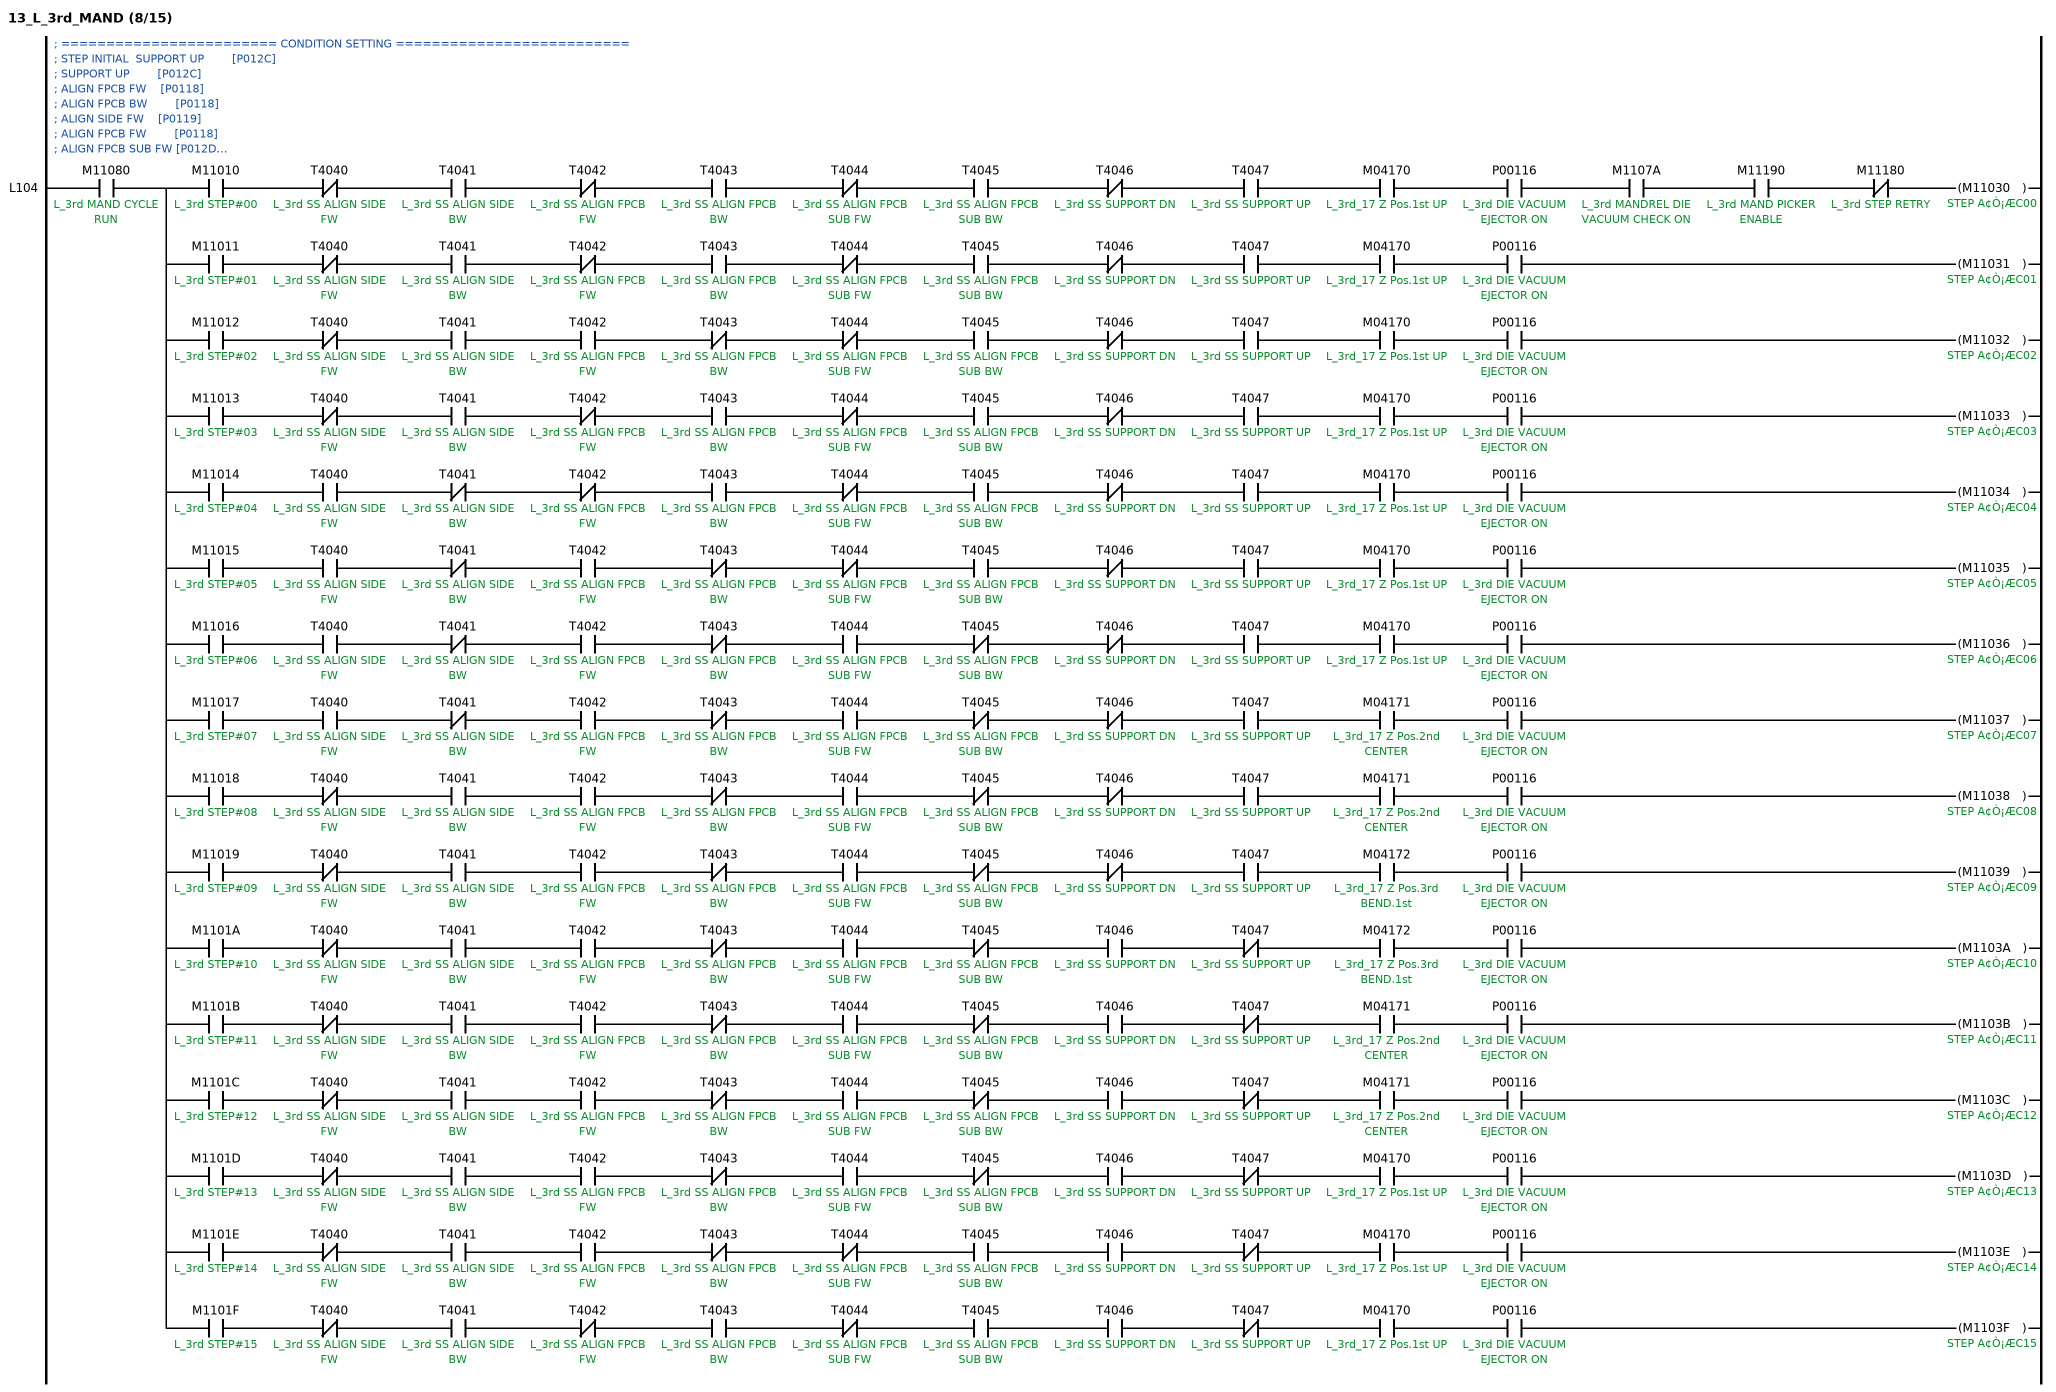
[picture p96: 13_L_3rd_MAND rungs L104-L104]
// ======================== CONDITION SETTING ==========================
; L104
LOAD      M11080	// L_3rd MAND CYCLE RUN
MPUSH
AND       M11010	// L_3rd STEP#00
AND NOT   T4040	// L_3rd SS ALIGN SIDE FW
AND       T4041	// L_3rd SS ALIGN SIDE BW
AND NOT   T4042	// L_3rd SS ALIGN FPCB FW
AND       T4043	// L_3rd SS ALIGN FPCB BW
AND NOT   T4044	// L_3rd SS ALIGN FPCB SUB FW
AND       T4045	// L_3rd SS ALIGN FPCB SUB BW
AND NOT   T4046	// L_3rd SS SUPPORT DN
AND       T4047	// L_3rd SS SUPPORT UP
AND       M04170	// L_3rd_17 Z Pos.1st UP
AND       P00116	// L_3rd DIE VACUUM EJECTOR ON
AND       M1107A	// L_3rd MANDREL DIE VACUUM CHECK ON
AND       M11190	// L_3rd MAND PICKER ENABLE
AND NOT   M11180	// L_3rd STEP RETRY
OUT       M11030	// STEP A¢Ò¡ÆC00
MLOAD
AND       M11011	// L_3rd STEP#01
AND NOT   T4040	// L_3rd SS ALIGN SIDE FW
AND       T4041	// L_3rd SS ALIGN SIDE BW
AND NOT   T4042	// L_3rd SS ALIGN FPCB FW
AND       T4043	// L_3rd SS ALIGN FPCB BW
AND NOT   T4044	// L_3rd SS ALIGN FPCB SUB FW
AND       T4045	// L_3rd SS ALIGN FPCB SUB BW
AND NOT   T4046	// L_3rd SS SUPPORT DN
AND       T4047	// L_3rd SS SUPPORT UP
AND       M04170	// L_3rd_17 Z Pos.1st UP
AND       P00116	// L_3rd DIE VACUUM EJECTOR ON
OUT       M11031	// STEP A¢Ò¡ÆC01
MLOAD
AND       M11012	// L_3rd STEP#02
AND NOT   T4040	// L_3rd SS ALIGN SIDE FW
AND       T4041	// L_3rd SS ALIGN SIDE BW
AND       T4042	// L_3rd SS ALIGN FPCB FW
AND NOT   T4043	// L_3rd SS ALIGN FPCB BW
AND NOT   T4044	// L_3rd SS ALIGN FPCB SUB FW
AND       T4045	// L_3rd SS ALIGN FPCB SUB BW
AND NOT   T4046	// L_3rd SS SUPPORT DN
AND       T4047	// L_3rd SS SUPPORT UP
AND       M04170	// L_3rd_17 Z Pos.1st UP
AND       P00116	// L_3rd DIE VACUUM EJECTOR ON
OUT       M11032	// STEP A¢Ò¡ÆC02
MLOAD
AND       M11013	// L_3rd STEP#03
AND NOT   T4040	// L_3rd SS ALIGN SIDE FW
AND       T4041	// L_3rd SS ALIGN SIDE BW
AND NOT   T4042	// L_3rd SS ALIGN FPCB FW
AND       T4043	// L_3rd SS ALIGN FPCB BW
AND NOT   T4044	// L_3rd SS ALIGN FPCB SUB FW
AND       T4045	// L_3rd SS ALIGN FPCB SUB BW
AND NOT   T4046	// L_3rd SS SUPPORT DN
AND       T4047	// L_3rd SS SUPPORT UP
AND       M04170	// L_3rd_17 Z Pos.1st UP
AND       P00116	// L_3rd DIE VACUUM EJECTOR ON
OUT       M11033	// STEP A¢Ò¡ÆC03
MLOAD
AND       M11014	// L_3rd STEP#04
AND       T4040	// L_3rd SS ALIGN SIDE FW
AND NOT   T4041	// L_3rd SS ALIGN SIDE BW
AND NOT   T4042	// L_3rd SS ALIGN FPCB FW
AND       T4043	// L_3rd SS ALIGN FPCB BW
AND NOT   T4044	// L_3rd SS ALIGN FPCB SUB FW
AND       T4045	// L_3rd SS ALIGN FPCB SUB BW
AND NOT   T4046	// L_3rd SS SUPPORT DN
AND       T4047	// L_3rd SS SUPPORT UP
AND       M04170	// L_3rd_17 Z Pos.1st UP
AND       P00116	// L_3rd DIE VACUUM EJECTOR ON
OUT       M11034	// STEP A¢Ò¡ÆC04
MLOAD
AND       M11015	// L_3rd STEP#05
AND       T4040	// L_3rd SS ALIGN SIDE FW
AND NOT   T4041	// L_3rd SS ALIGN SIDE BW
AND       T4042	// L_3rd SS ALIGN FPCB FW
AND NOT   T4043	// L_3rd SS ALIGN FPCB BW
AND NOT   T4044	// L_3rd SS ALIGN FPCB SUB FW
AND       T4045	// L_3rd SS ALIGN FPCB SUB BW
AND NOT   T4046	// L_3rd SS SUPPORT DN
AND       T4047	// L_3rd SS SUPPORT UP
AND       M04170	// L_3rd_17 Z Pos.1st UP
AND       P00116	// L_3rd DIE VACUUM EJECTOR ON
OUT       M11035	// STEP A¢Ò¡ÆC05
MLOAD
AND       M11016	// L_3rd STEP#06
AND       T4040	// L_3rd SS ALIGN SIDE FW
AND NOT   T4041	// L_3rd SS ALIGN SIDE BW
AND       T4042	// L_3rd SS ALIGN FPCB FW
AND NOT   T4043	// L_3rd SS ALIGN FPCB BW
AND       T4044	// L_3rd SS ALIGN FPCB SUB FW
AND NOT   T4045	// L_3rd SS ALIGN FPCB SUB BW
AND NOT   T4046	// L_3rd SS SUPPORT DN
AND       T4047	// L_3rd SS SUPPORT UP
AND       M04170	// L_3rd_17 Z Pos.1st UP
AND       P00116	// L_3rd DIE VACUUM EJECTOR ON
OUT       M11036	// STEP A¢Ò¡ÆC06
MLOAD
AND       M11017	// L_3rd STEP#07
AND       T4040	// L_3rd SS ALIGN SIDE FW
AND NOT   T4041	// L_3rd SS ALIGN SIDE BW
AND       T4042	// L_3rd SS ALIGN FPCB FW
AND NOT   T4043	// L_3rd SS ALIGN FPCB BW
AND       T4044	// L_3rd SS ALIGN FPCB SUB FW
AND NOT   T4045	// L_3rd SS ALIGN FPCB SUB BW
AND NOT   T4046	// L_3rd SS SUPPORT DN
AND       T4047	// L_3rd SS SUPPORT UP
AND       M04171	// L_3rd_17 Z Pos.2nd CENTER
AND       P00116	// L_3rd DIE VACUUM EJECTOR ON
OUT       M11037	// STEP A¢Ò¡ÆC07
MLOAD
AND       M11018	// L_3rd STEP#08
AND NOT   T4040	// L_3rd SS ALIGN SIDE FW
AND       T4041	// L_3rd SS ALIGN SIDE BW
AND       T4042	// L_3rd SS ALIGN FPCB FW
AND NOT   T4043	// L_3rd SS ALIGN FPCB BW
AND       T4044	// L_3rd SS ALIGN FPCB SUB FW
AND NOT   T4045	// L_3rd SS ALIGN FPCB SUB BW
AND NOT   T4046	// L_3rd SS SUPPORT DN
AND       T4047	// L_3rd SS SUPPORT UP
AND       M04171	// L_3rd_17 Z Pos.2nd CENTER
AND       P00116	// L_3rd DIE VACUUM EJECTOR ON
OUT       M11038	// STEP A¢Ò¡ÆC08
MLOAD
AND       M11019	// L_3rd STEP#09
AND NOT   T4040	// L_3rd SS ALIGN SIDE FW
AND       T4041	// L_3rd SS ALIGN SIDE BW
AND       T4042	// L_3rd SS ALIGN FPCB FW
AND NOT   T4043	// L_3rd SS ALIGN FPCB BW
AND       T4044	// L_3rd SS ALIGN FPCB SUB FW
AND NOT   T4045	// L_3rd SS ALIGN FPCB SUB BW
AND NOT   T4046	// L_3rd SS SUPPORT DN
AND       T4047	// L_3rd SS SUPPORT UP
AND       M04172	// L_3rd_17 Z Pos.3rd BEND.1st
AND       P00116	// L_3rd DIE VACUUM EJECTOR ON
OUT       M11039	// STEP A¢Ò¡ÆC09
MLOAD
AND       M1101A	// L_3rd STEP#10
AND NOT   T4040	// L_3rd SS ALIGN SIDE FW
AND       T4041	// L_3rd SS ALIGN SIDE BW
AND       T4042	// L_3rd SS ALIGN FPCB FW
AND NOT   T4043	// L_3rd SS ALIGN FPCB BW
AND       T4044	// L_3rd SS ALIGN FPCB SUB FW
AND NOT   T4045	// L_3rd SS ALIGN FPCB SUB BW
AND       T4046	// L_3rd SS SUPPORT DN
AND NOT   T4047	// L_3rd SS SUPPORT UP
AND       M04172	// L_3rd_17 Z Pos.3rd BEND.1st
AND       P00116	// L_3rd DIE VACUUM EJECTOR ON
OUT       M1103A	// STEP A¢Ò¡ÆC10
MLOAD
AND       M1101B	// L_3rd STEP#11
AND NOT   T4040	// L_3rd SS ALIGN SIDE FW
AND       T4041	// L_3rd SS ALIGN SIDE BW
AND       T4042	// L_3rd SS ALIGN FPCB FW
AND NOT   T4043	// L_3rd SS ALIGN FPCB BW
AND       T4044	// L_3rd SS ALIGN FPCB SUB FW
AND NOT   T4045	// L_3rd SS ALIGN FPCB SUB BW
AND       T4046	// L_3rd SS SUPPORT DN
AND NOT   T4047	// L_3rd SS SUPPORT UP
AND       M04171	// L_3rd_17 Z Pos.2nd CENTER
AND       P00116	// L_3rd DIE VACUUM EJECTOR ON
OUT       M1103B	// STEP A¢Ò¡ÆC11
MLOAD
AND       M1101C	// L_3rd STEP#12
AND NOT   T4040	// L_3rd SS ALIGN SIDE FW
AND       T4041	// L_3rd SS ALIGN SIDE BW
AND       T4042	// L_3rd SS ALIGN FPCB FW
AND NOT   T4043	// L_3rd SS ALIGN FPCB BW
AND       T4044	// L_3rd SS ALIGN FPCB SUB FW
AND NOT   T4045	// L_3rd SS ALIGN FPCB SUB BW
AND       T4046	// L_3rd SS SUPPORT DN
AND NOT   T4047	// L_3rd SS SUPPORT UP
AND       M04171	// L_3rd_17 Z Pos.2nd CENTER
AND       P00116	// L_3rd DIE VACUUM EJECTOR ON
OUT       M1103C	// STEP A¢Ò¡ÆC12
MLOAD
AND       M1101D	// L_3rd STEP#13
AND NOT   T4040	// L_3rd SS ALIGN SIDE FW
AND       T4041	// L_3rd SS ALIGN SIDE BW
AND       T4042	// L_3rd SS ALIGN FPCB FW
AND NOT   T4043	// L_3rd SS ALIGN FPCB BW
AND       T4044	// L_3rd SS ALIGN FPCB SUB FW
AND NOT   T4045	// L_3rd SS ALIGN FPCB SUB BW
AND       T4046	// L_3rd SS SUPPORT DN
AND NOT   T4047	// L_3rd SS SUPPORT UP
AND       M04170	// L_3rd_17 Z Pos.1st UP
AND       P00116	// L_3rd DIE VACUUM EJECTOR ON
OUT       M1103D	// STEP A¢Ò¡ÆC13
MLOAD
AND       M1101E	// L_3rd STEP#14
AND NOT   T4040	// L_3rd SS ALIGN SIDE FW
AND       T4041	// L_3rd SS ALIGN SIDE BW
AND       T4042	// L_3rd SS ALIGN FPCB FW
AND NOT   T4043	// L_3rd SS ALIGN FPCB BW
AND NOT   T4044	// L_3rd SS ALIGN FPCB SUB FW
AND       T4045	// L_3rd SS ALIGN FPCB SUB BW
AND       T4046	// L_3rd SS SUPPORT DN
AND NOT   T4047	// L_3rd SS SUPPORT UP
AND       M04170	// L_3rd_17 Z Pos.1st UP
AND       P00116	// L_3rd DIE VACUUM EJECTOR ON
OUT       M1103E	// STEP A¢Ò¡ÆC14
MPOP
AND       M1101F	// L_3rd STEP#15
AND NOT   T4040	// L_3rd SS ALIGN SIDE FW
AND       T4041	// L_3rd SS ALIGN SIDE BW
AND NOT   T4042	// L_3rd SS ALIGN FPCB FW
AND       T4043	// L_3rd SS ALIGN FPCB BW
AND NOT   T4044	// L_3rd SS ALIGN FPCB SUB FW
AND       T4045	// L_3rd SS ALIGN FPCB SUB BW
AND       T4046	// L_3rd SS SUPPORT DN
AND NOT   T4047	// L_3rd SS SUPPORT UP
AND       M04170	// L_3rd_17 Z Pos.1st UP
AND       P00116	// L_3rd DIE VACUUM EJECTOR ON
OUT       M1103F	// STEP A¢Ò¡ÆC15
// output comment: STEP INITIAL  SUPPORT UP        [P012C]
// output comment: SUPPORT UP        [P012C]
// output comment: ALIGN FPCB FW    [P0118]
// output comment: ALIGN FPCB BW        [P0118]
// output comment: ALIGN SIDE FW    [P0119]
// output comment: ALIGN FPCB FW        [P0118]
// output comment: ALIGN FPCB SUB FW [P012D]
// output comment: L_3rd_17 Z Pos.2nd CENTER >
// output comment: ALIGN SIDE BW      [P0119]
// output comment: L_3rd_17 Z Pos.3rd BEND.1st >
// output comment: SUPPORT DN      [P012C]
// output comment: L_3rd_17 Z Pos.2nd CENTER >
// output comment: L_3rd_17 Z Pos.1st      UP >
// output comment: ALIGN FPCB SUB BW [P012D]
// output comment: ALIGN FPCB BW    [P0118]

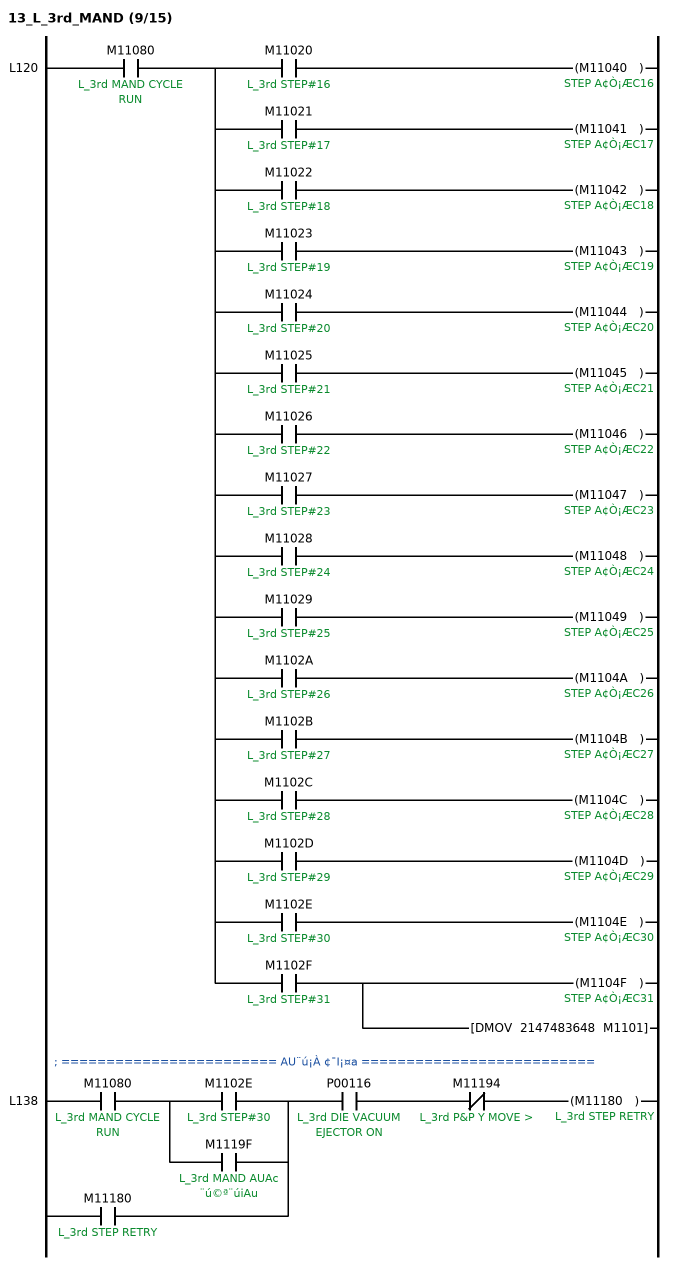
; L120
LOAD      M11080	// L_3rd MAND CYCLE RUN
MPUSH
AND       M11020	// L_3rd STEP#16
OUT       M11040	// STEP A¢Ò¡ÆC16
MLOAD
AND       M11021	// L_3rd STEP#17
OUT       M11041	// STEP A¢Ò¡ÆC17
MLOAD
AND       M11022	// L_3rd STEP#18
OUT       M11042	// STEP A¢Ò¡ÆC18
MLOAD
AND       M11023	// L_3rd STEP#19
OUT       M11043	// STEP A¢Ò¡ÆC19
MLOAD
AND       M11024	// L_3rd STEP#20
OUT       M11044	// STEP A¢Ò¡ÆC20
MLOAD
AND       M11025	// L_3rd STEP#21
OUT       M11045	// STEP A¢Ò¡ÆC21
MLOAD
AND       M11026	// L_3rd STEP#22
OUT       M11046	// STEP A¢Ò¡ÆC22
MLOAD
AND       M11027	// L_3rd STEP#23
OUT       M11047	// STEP A¢Ò¡ÆC23
MLOAD
AND       M11028	// L_3rd STEP#24
OUT       M11048	// STEP A¢Ò¡ÆC24
MLOAD
AND       M11029	// L_3rd STEP#25
OUT       M11049	// STEP A¢Ò¡ÆC25
MLOAD
AND       M1102A	// L_3rd STEP#26
OUT       M1104A	// STEP A¢Ò¡ÆC26
MLOAD
AND       M1102B	// L_3rd STEP#27
OUT       M1104B	// STEP A¢Ò¡ÆC27
MLOAD
AND       M1102C	// L_3rd STEP#28
OUT       M1104C	// STEP A¢Ò¡ÆC28
MLOAD
AND       M1102D	// L_3rd STEP#29
OUT       M1104D	// STEP A¢Ò¡ÆC29
MLOAD
AND       M1102E	// L_3rd STEP#30
OUT       M1104E	// STEP A¢Ò¡ÆC30
MPOP
AND       M1102F	// L_3rd STEP#31
OUT       M1104F	// STEP A¢Ò¡ÆC31
DMOV      2147483648 M1101
// ======================== AU¨ú¡À ¢¯I¡¤a ==========================
; L138
LOAD      M11080	// L_3rd MAND CYCLE RUN
LOAD      M1102E	// L_3rd STEP#30
OR        M1119F	// L_3rd MAND AUAc ¨ú©ª¨úiAu
AND LOAD
OR        M11180	// L_3rd STEP RETRY
AND       P00116	// L_3rd DIE VACUUM EJECTOR ON
AND NOT   M11194	// L_3rd P&P Y MOVE >
OUT       M11180	// L_3rd STEP RETRY

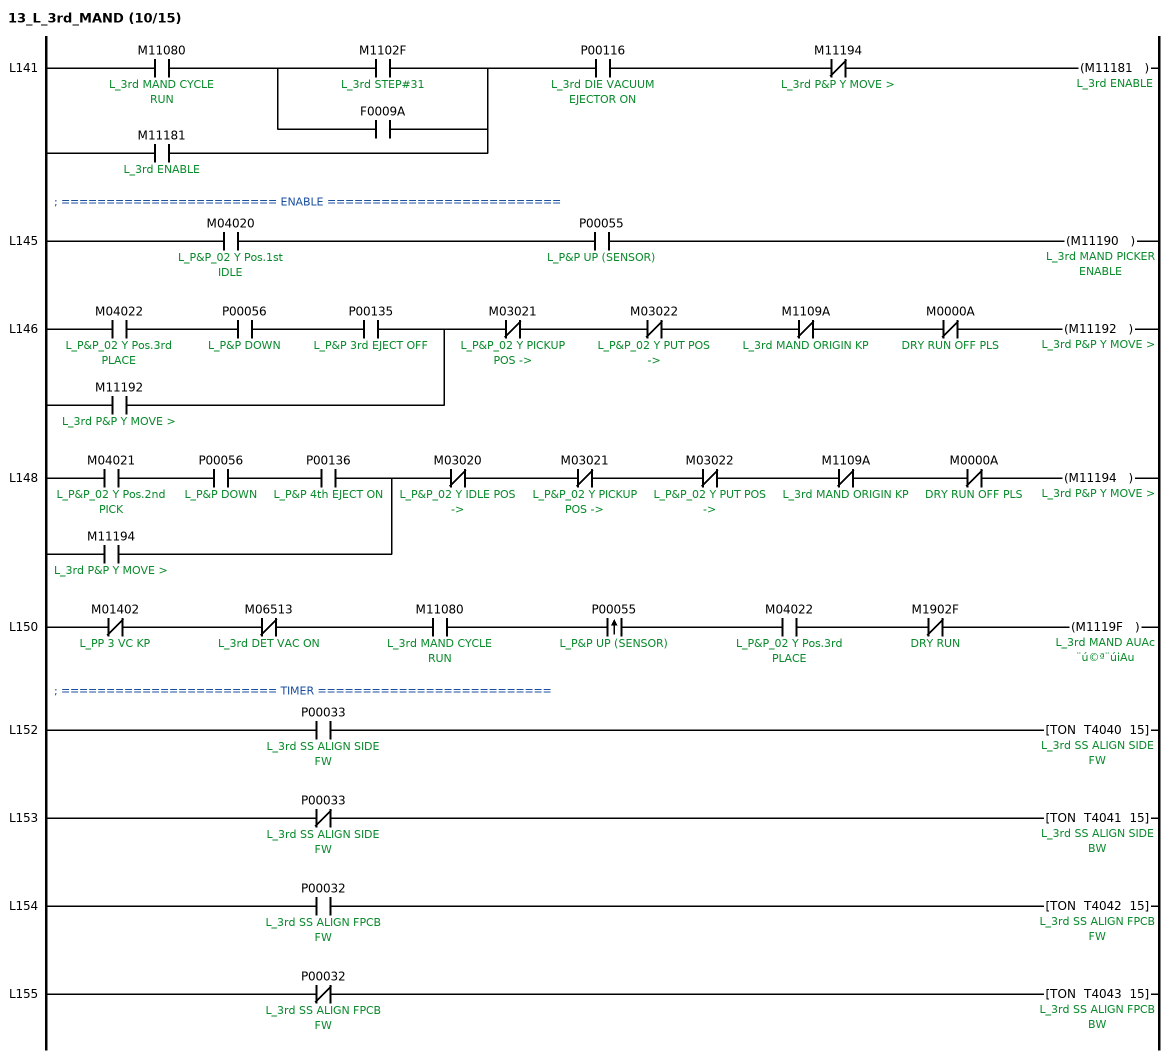
; L141
LOAD      M11080	// L_3rd MAND CYCLE RUN
LOAD      M1102F	// L_3rd STEP#31
OR        F0009A
AND LOAD
OR        M11181	// L_3rd ENABLE
AND       P00116	// L_3rd DIE VACUUM EJECTOR ON
AND NOT   M11194	// L_3rd P&P Y MOVE >
OUT       M11181	// L_3rd ENABLE
// ======================== ENABLE ==========================
; L145
LOAD      M04020	// L_P&P_02 Y Pos.1st IDLE
AND       P00055	// L_P&P UP (SENSOR)
OUT       M11190	// L_3rd MAND PICKER ENABLE
; L146
LOAD      M04022	// L_P&P_02 Y Pos.3rd PLACE
AND       P00056	// L_P&P DOWN
AND       P00135	// L_P&P 3rd EJECT OFF
OR        M11192	// L_3rd P&P Y MOVE >
AND NOT   M03021	// L_P&P_02 Y PICKUP POS ->
AND NOT   M03022	// L_P&P_02 Y PUT POS ->
AND NOT   M1109A	// L_3rd MAND ORIGIN KP
AND NOT   M0000A	// DRY RUN OFF PLS
OUT       M11192	// L_3rd P&P Y MOVE >
; L148
LOAD      M04021	// L_P&P_02 Y Pos.2nd PICK
AND       P00056	// L_P&P DOWN
AND       P00136	// L_P&P 4th EJECT ON
OR        M11194	// L_3rd P&P Y MOVE >
AND NOT   M03020	// L_P&P_02 Y IDLE POS ->
AND NOT   M03021	// L_P&P_02 Y PICKUP POS ->
AND NOT   M03022	// L_P&P_02 Y PUT POS ->
AND NOT   M1109A	// L_3rd MAND ORIGIN KP
AND NOT   M0000A	// DRY RUN OFF PLS
OUT       M11194	// L_3rd P&P Y MOVE >
; L150
LOAD NOT  M01402	// L_PP 3 VC KP
AND NOT   M06513	// L_3rd DET VAC ON
AND       M11080	// L_3rd MAND CYCLE RUN
ANDP      P00055	// L_P&P UP (SENSOR)
AND       M04022	// L_P&P_02 Y Pos.3rd PLACE
AND NOT   M1902F	// DRY RUN
OUT       M1119F	// L_3rd MAND AUAc ¨ú©ª¨úiAu
// ======================== TIMER ==========================
; L152
LOAD      P00033	// L_3rd SS ALIGN SIDE FW
TON       T4040 15	// L_3rd SS ALIGN SIDE FW
; L153
LOAD NOT  P00033	// L_3rd SS ALIGN SIDE FW
TON       T4041 15	// L_3rd SS ALIGN SIDE BW
; L154
LOAD      P00032	// L_3rd SS ALIGN FPCB FW
TON       T4042 15	// L_3rd SS ALIGN FPCB FW
; L155
LOAD NOT  P00032	// L_3rd SS ALIGN FPCB FW
TON       T4043 15	// L_3rd SS ALIGN FPCB BW

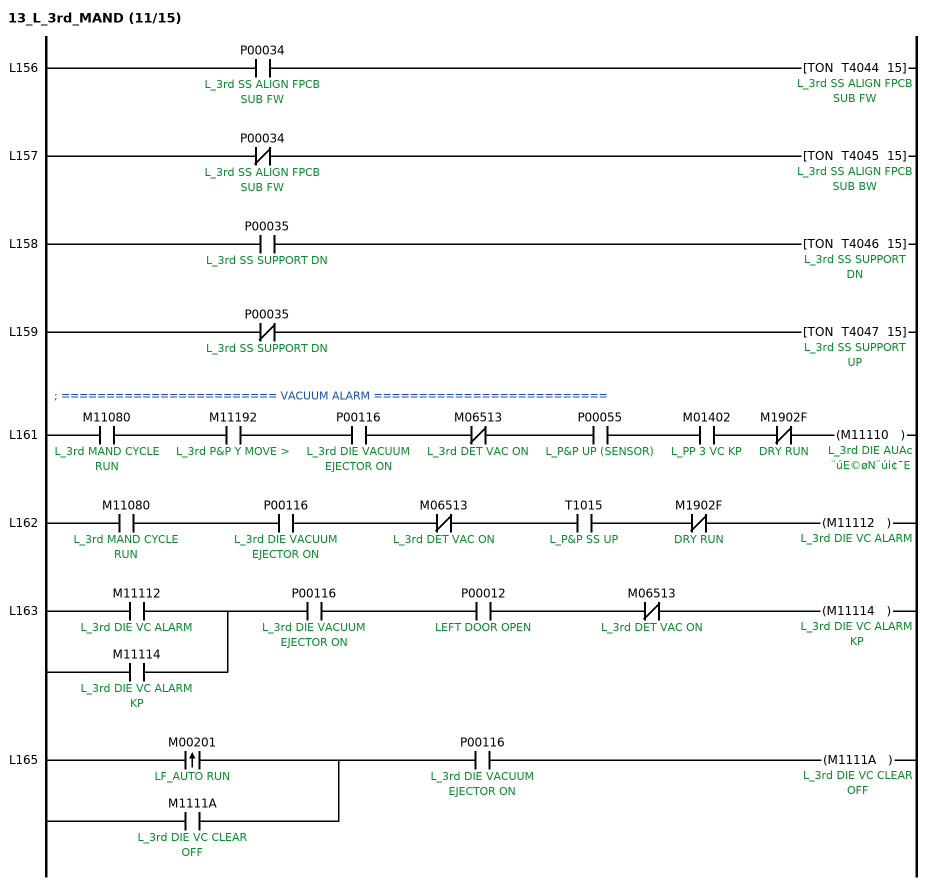
; L156
LOAD      P00034	// L_3rd SS ALIGN FPCB SUB FW
TON       T4044 15	// L_3rd SS ALIGN FPCB SUB FW
; L157
LOAD NOT  P00034	// L_3rd SS ALIGN FPCB SUB FW
TON       T4045 15	// L_3rd SS ALIGN FPCB SUB BW
; L158
LOAD      P00035	// L_3rd SS SUPPORT DN
TON       T4046 15	// L_3rd SS SUPPORT DN
; L159
LOAD NOT  P00035	// L_3rd SS SUPPORT DN
TON       T4047 15	// L_3rd SS SUPPORT UP
// ======================== VACUUM ALARM ==========================
; L161
LOAD      M11080	// L_3rd MAND CYCLE RUN
AND       M11192	// L_3rd P&P Y MOVE >
AND       P00116	// L_3rd DIE VACUUM EJECTOR ON
AND NOT   M06513	// L_3rd DET VAC ON
AND       P00055	// L_P&P UP (SENSOR)
AND       M01402	// L_PP 3 VC KP
AND NOT   M1902F	// DRY RUN
OUT       M11110	// L_3rd DIE AUAc ¨úE©øN¨úi¢¯E
; L162
LOAD      M11080	// L_3rd MAND CYCLE RUN
AND       P00116	// L_3rd DIE VACUUM EJECTOR ON
AND NOT   M06513	// L_3rd DET VAC ON
AND       T1015	// L_P&P SS UP
AND NOT   M1902F	// DRY RUN
OUT       M11112	// L_3rd DIE VC ALARM
; L163
LOAD      M11112	// L_3rd DIE VC ALARM
OR        M11114	// L_3rd DIE VC ALARM KP
AND       P00116	// L_3rd DIE VACUUM EJECTOR ON
AND       P00012	// LEFT DOOR OPEN
AND NOT   M06513	// L_3rd DET VAC ON
OUT       M11114	// L_3rd DIE VC ALARM KP
; L165
LOADP     M00201	// LF_AUTO RUN
OR        M1111A	// L_3rd DIE VC CLEAR OFF
AND       P00116	// L_3rd DIE VACUUM EJECTOR ON
OUT       M1111A	// L_3rd DIE VC CLEAR OFF

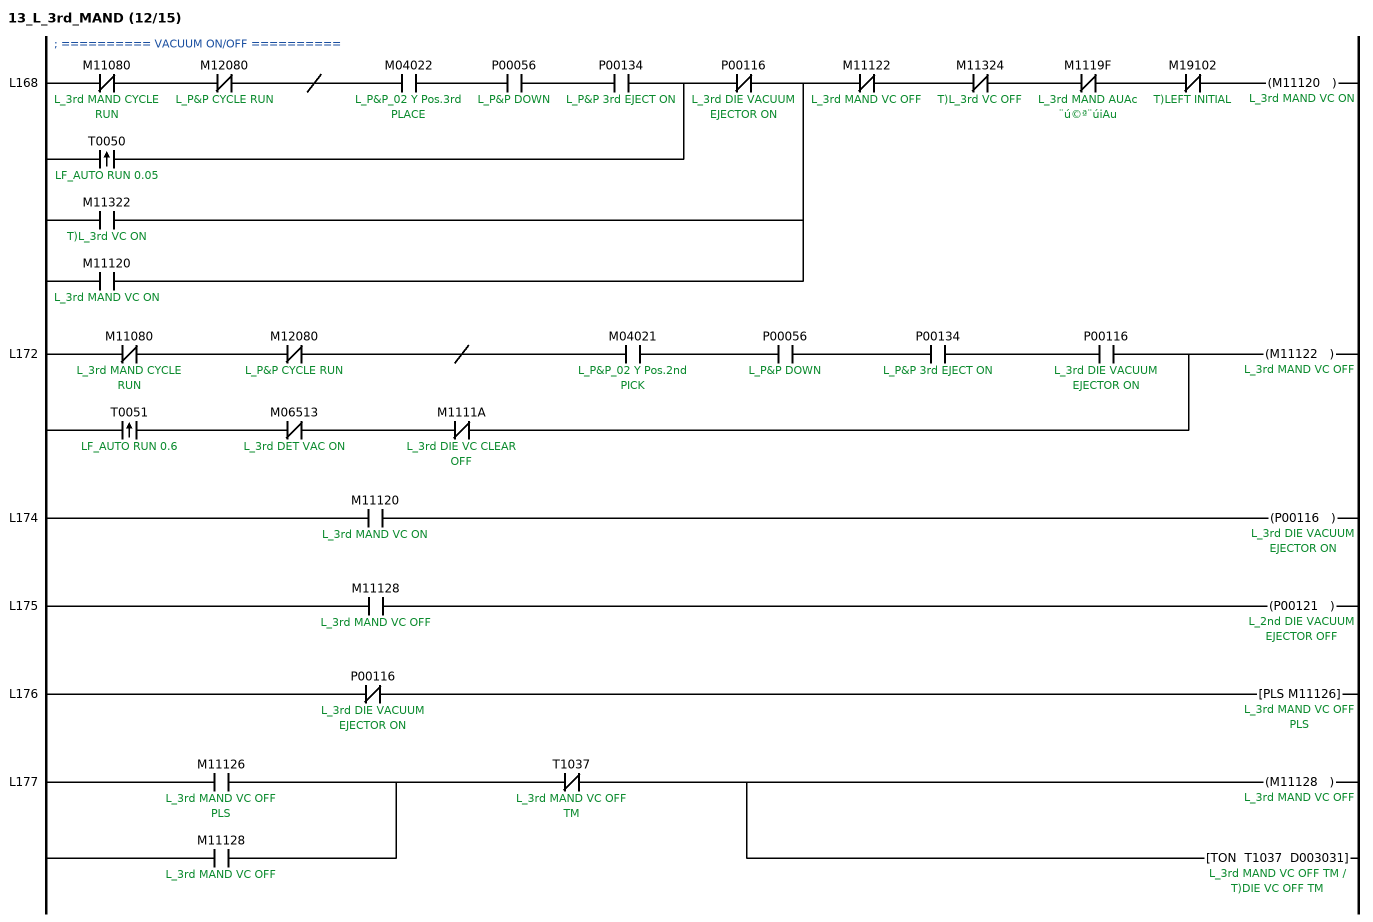
// ========== VACUUM ON/OFF ==========
; L168
LOAD NOT  M11080	// L_3rd MAND CYCLE RUN
AND NOT   M12080	// L_P&P CYCLE RUN
NOT
AND       M04022	// L_P&P_02 Y Pos.3rd PLACE
AND       P00056	// L_P&P DOWN
AND       P00134	// L_P&P 3rd EJECT ON
ORP       T0050	// LF_AUTO RUN 0.05
AND NOT   P00116	// L_3rd DIE VACUUM EJECTOR ON
OR        M11322	// T)L_3rd VC ON
OR        M11120	// L_3rd MAND VC ON
AND NOT   M11122	// L_3rd MAND VC OFF
AND NOT   M11324	// T)L_3rd VC OFF
AND NOT   M1119F	// L_3rd MAND AUAc ¨ú©ª¨úiAu
AND NOT   M19102	// T)LEFT INITIAL
OUT       M11120	// L_3rd MAND VC ON
; L172
LOAD NOT  M11080	// L_3rd MAND CYCLE RUN
AND NOT   M12080	// L_P&P CYCLE RUN
NOT
AND       M04021	// L_P&P_02 Y Pos.2nd PICK
AND       P00056	// L_P&P DOWN
AND       P00134	// L_P&P 3rd EJECT ON
AND       P00116	// L_3rd DIE VACUUM EJECTOR ON
LOADP     T0051	// LF_AUTO RUN 0.6
AND NOT   M06513	// L_3rd DET VAC ON
AND NOT   M1111A	// L_3rd DIE VC CLEAR OFF
OR LOAD
OUT       M11122	// L_3rd MAND VC OFF
; L174
LOAD      M11120	// L_3rd MAND VC ON
OUT       P00116	// L_3rd DIE VACUUM EJECTOR ON
; L175
LOAD      M11128	// L_3rd MAND VC OFF
OUT       P00121	// L_2nd DIE VACUUM EJECTOR OFF
; L176
LOAD NOT  P00116	// L_3rd DIE VACUUM EJECTOR ON
OUTP      M11126	// L_3rd MAND VC OFF PLS
; L177
LOAD      M11126	// L_3rd MAND VC OFF PLS
OR        M11128	// L_3rd MAND VC OFF
AND NOT   T1037	// L_3rd MAND VC OFF TM
OUT       M11128	// L_3rd MAND VC OFF
TON       T1037 D003031	// L_3rd MAND VC OFF TM / T)DIE VC OFF TM

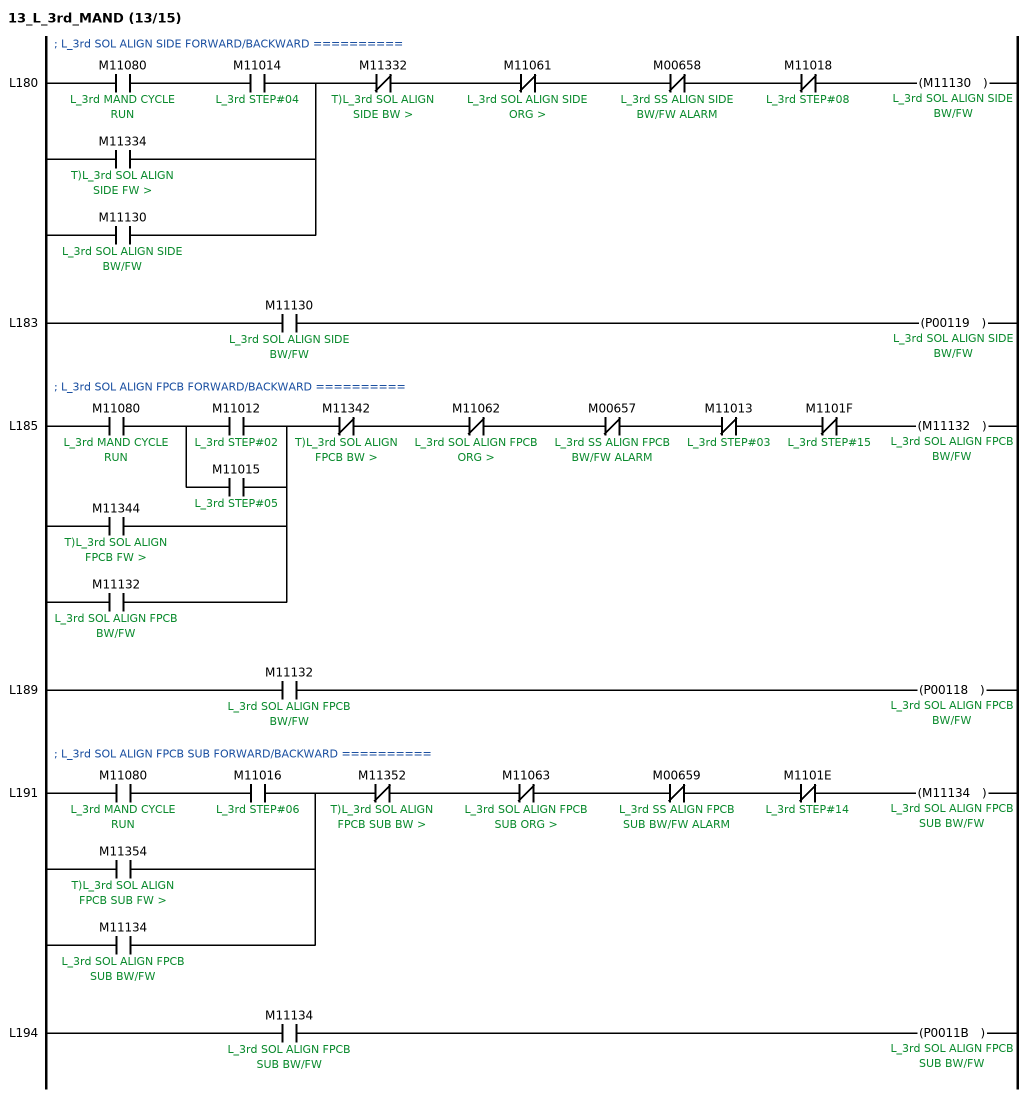
// L_3rd SOL ALIGN SIDE FORWARD/BACKWARD ==========
; L180
LOAD      M11080	// L_3rd MAND CYCLE RUN
AND       M11014	// L_3rd STEP#04
OR        M11334	// T)L_3rd SOL ALIGN SIDE FW >
OR        M11130	// L_3rd SOL ALIGN SIDE BW/FW
AND NOT   M11332	// T)L_3rd SOL ALIGN SIDE BW >
AND NOT   M11061	// L_3rd SOL ALIGN SIDE ORG >
AND NOT   M00658	// L_3rd SS ALIGN SIDE BW/FW ALARM
AND NOT   M11018	// L_3rd STEP#08
OUT       M11130	// L_3rd SOL ALIGN SIDE BW/FW
; L183
LOAD      M11130	// L_3rd SOL ALIGN SIDE BW/FW
OUT       P00119	// L_3rd SOL ALIGN SIDE BW/FW
// L_3rd SOL ALIGN FPCB FORWARD/BACKWARD ==========
; L185
LOAD      M11080	// L_3rd MAND CYCLE RUN
LOAD      M11012	// L_3rd STEP#02
OR        M11015	// L_3rd STEP#05
AND LOAD
OR        M11344	// T)L_3rd SOL ALIGN FPCB FW >
OR        M11132	// L_3rd SOL ALIGN FPCB BW/FW
AND NOT   M11342	// T)L_3rd SOL ALIGN FPCB BW >
AND NOT   M11062	// L_3rd SOL ALIGN FPCB ORG >
AND NOT   M00657	// L_3rd SS ALIGN FPCB BW/FW ALARM
AND NOT   M11013	// L_3rd STEP#03
AND NOT   M1101F	// L_3rd STEP#15
OUT       M11132	// L_3rd SOL ALIGN FPCB BW/FW
; L189
LOAD      M11132	// L_3rd SOL ALIGN FPCB BW/FW
OUT       P00118	// L_3rd SOL ALIGN FPCB BW/FW
// L_3rd SOL ALIGN FPCB SUB FORWARD/BACKWARD ==========
; L191
LOAD      M11080	// L_3rd MAND CYCLE RUN
AND       M11016	// L_3rd STEP#06
OR        M11354	// T)L_3rd SOL ALIGN FPCB SUB FW >
OR        M11134	// L_3rd SOL ALIGN FPCB SUB BW/FW
AND NOT   M11352	// T)L_3rd SOL ALIGN FPCB SUB BW >
AND NOT   M11063	// L_3rd SOL ALIGN FPCB SUB ORG >
AND NOT   M00659	// L_3rd SS ALIGN FPCB SUB BW/FW ALARM
AND NOT   M1101E	// L_3rd STEP#14
OUT       M11134	// L_3rd SOL ALIGN FPCB SUB BW/FW
; L194
LOAD      M11134	// L_3rd SOL ALIGN FPCB SUB BW/FW
OUT       P0011B	// L_3rd SOL ALIGN FPCB SUB BW/FW

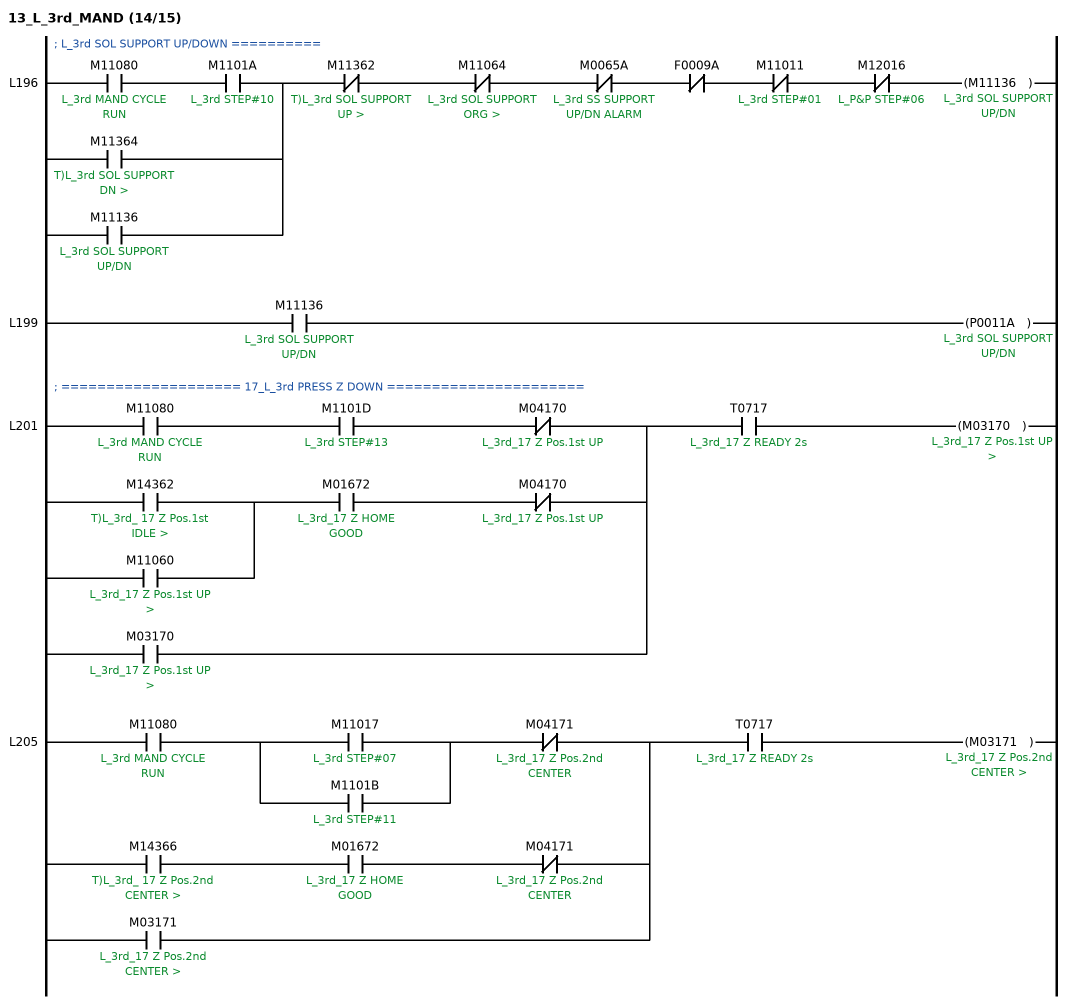
// L_3rd SOL SUPPORT UP/DOWN ==========
; L196
LOAD      M11080	// L_3rd MAND CYCLE RUN
AND       M1101A	// L_3rd STEP#10
OR        M11364	// T)L_3rd SOL SUPPORT DN >
OR        M11136	// L_3rd SOL SUPPORT UP/DN
AND NOT   M11362	// T)L_3rd SOL SUPPORT UP >
AND NOT   M11064	// L_3rd SOL SUPPORT ORG >
AND NOT   M0065A	// L_3rd SS SUPPORT UP/DN ALARM
AND NOT   F0009A
AND NOT   M11011	// L_3rd STEP#01
AND NOT   M12016	// L_P&P STEP#06
OUT       M11136	// L_3rd SOL SUPPORT UP/DN
; L199
LOAD      M11136	// L_3rd SOL SUPPORT UP/DN
OUT       P0011A	// L_3rd SOL SUPPORT UP/DN
// ==================== 17_L_3rd PRESS Z DOWN ======================
; L201
LOAD      M11080	// L_3rd MAND CYCLE RUN
AND       M1101D	// L_3rd STEP#13
AND NOT   M04170	// L_3rd_17 Z Pos.1st UP
LOAD      M14362	// T)L_3rd_ 17 Z Pos.1st IDLE >
OR        M11060	// L_3rd_17 Z Pos.1st UP >
AND       M01672	// L_3rd_17 Z HOME GOOD
AND NOT   M04170	// L_3rd_17 Z Pos.1st UP
OR LOAD
OR        M03170	// L_3rd_17 Z Pos.1st UP >
AND       T0717	// L_3rd_17 Z READY 2s
OUT       M03170	// L_3rd_17 Z Pos.1st UP >
; L205
LOAD      M11080	// L_3rd MAND CYCLE RUN
LOAD      M11017	// L_3rd STEP#07
OR        M1101B	// L_3rd STEP#11
AND LOAD
AND NOT   M04171	// L_3rd_17 Z Pos.2nd CENTER
LOAD      M14366	// T)L_3rd_ 17 Z Pos.2nd CENTER >
AND       M01672	// L_3rd_17 Z HOME GOOD
AND NOT   M04171	// L_3rd_17 Z Pos.2nd CENTER
OR LOAD
OR        M03171	// L_3rd_17 Z Pos.2nd CENTER >
AND       T0717	// L_3rd_17 Z READY 2s
OUT       M03171	// L_3rd_17 Z Pos.2nd CENTER >

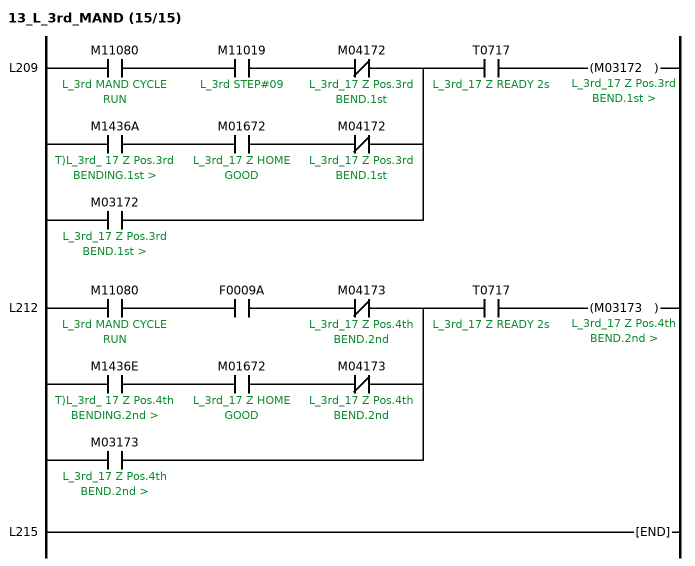
; L209
LOAD      M11080	// L_3rd MAND CYCLE RUN
AND       M11019	// L_3rd STEP#09
AND NOT   M04172	// L_3rd_17 Z Pos.3rd BEND.1st
LOAD      M1436A	// T)L_3rd_ 17 Z Pos.3rd BENDING.1st >
AND       M01672	// L_3rd_17 Z HOME GOOD
AND NOT   M04172	// L_3rd_17 Z Pos.3rd BEND.1st
OR LOAD
OR        M03172	// L_3rd_17 Z Pos.3rd BEND.1st >
AND       T0717	// L_3rd_17 Z READY 2s
OUT       M03172	// L_3rd_17 Z Pos.3rd BEND.1st >
; L212
LOAD      M11080	// L_3rd MAND CYCLE RUN
AND       F0009A
AND NOT   M04173	// L_3rd_17 Z Pos.4th BEND.2nd
LOAD      M1436E	// T)L_3rd_ 17 Z Pos.4th BENDING.2nd >
AND       M01672	// L_3rd_17 Z HOME GOOD
AND NOT   M04173	// L_3rd_17 Z Pos.4th BEND.2nd
OR LOAD
OR        M03173	// L_3rd_17 Z Pos.4th BEND.2nd >
AND       T0717	// L_3rd_17 Z READY 2s
OUT       M03173	// L_3rd_17 Z Pos.4th BEND.2nd >
; L215
END

PROGRAM 14_L_TOOL (task: ½ºÄµ ÇÁ·Î±×·¥)

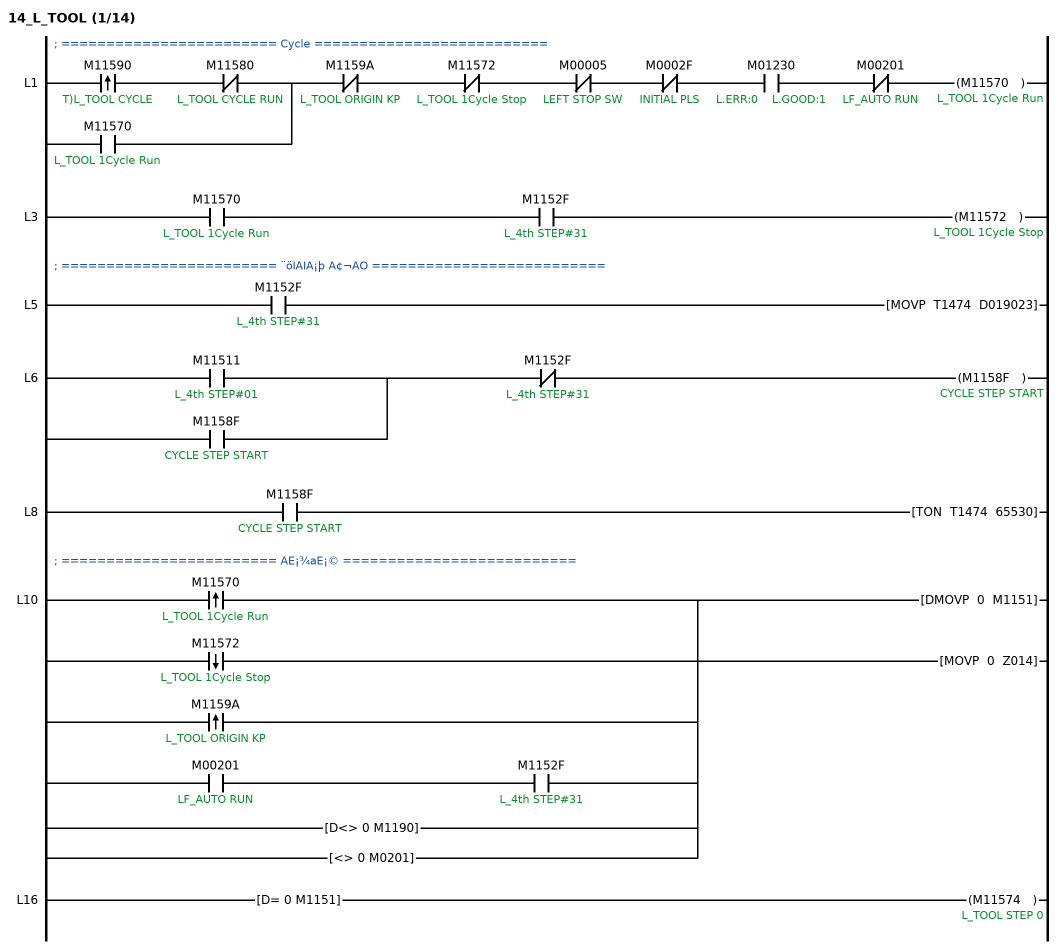
// ======================== Cycle ==========================
; L1
LOADP     M11590	// T)L_TOOL CYCLE
AND NOT   M11580	// L_TOOL CYCLE RUN
OR        M11570	// L_TOOL 1Cycle Run
AND NOT   M1159A	// L_TOOL ORIGIN KP
AND NOT   M11572	// L_TOOL 1Cycle Stop
AND NOT   M00005	// LEFT STOP SW
AND NOT   M0002F	// INITIAL PLS
AND       M01230	// L.ERR:0    L.GOOD:1
AND NOT   M00201	// LF_AUTO RUN
OUT       M11570	// L_TOOL 1Cycle Run
; L3
LOAD      M11570	// L_TOOL 1Cycle Run
AND       M1152F	// L_4th STEP#31
OUT       M11572	// L_TOOL 1Cycle Stop
// ======================== ¨öIAIA¡þ A¢¬AO ==========================
; L5
LOAD      M1152F	// L_4th STEP#31
MOVP      T1474 D019023
; L6
LOAD      M11511	// L_4th STEP#01
OR        M1158F	// CYCLE STEP START
AND NOT   M1152F	// L_4th STEP#31
OUT       M1158F	// CYCLE STEP START
; L8
LOAD      M1158F	// CYCLE STEP START
TON       T1474 65530
// ======================== AE¡¾aE¡© ==========================
; L10
LOADP     M11570	// L_TOOL 1Cycle Run
ORN       M11572	// L_TOOL 1Cycle Stop
ORP       M1159A	// L_TOOL ORIGIN KP
LOAD      M00201	// LF_AUTO RUN
AND       M1152F	// L_4th STEP#31
OR LOAD
ORD<>     0 M1190
OR<>      0 M0201
DMOVP     0 M1151
MOVP      0 Z014
; L16
LOADD=    0 M1151
OUT       M11574	// L_TOOL STEP 0

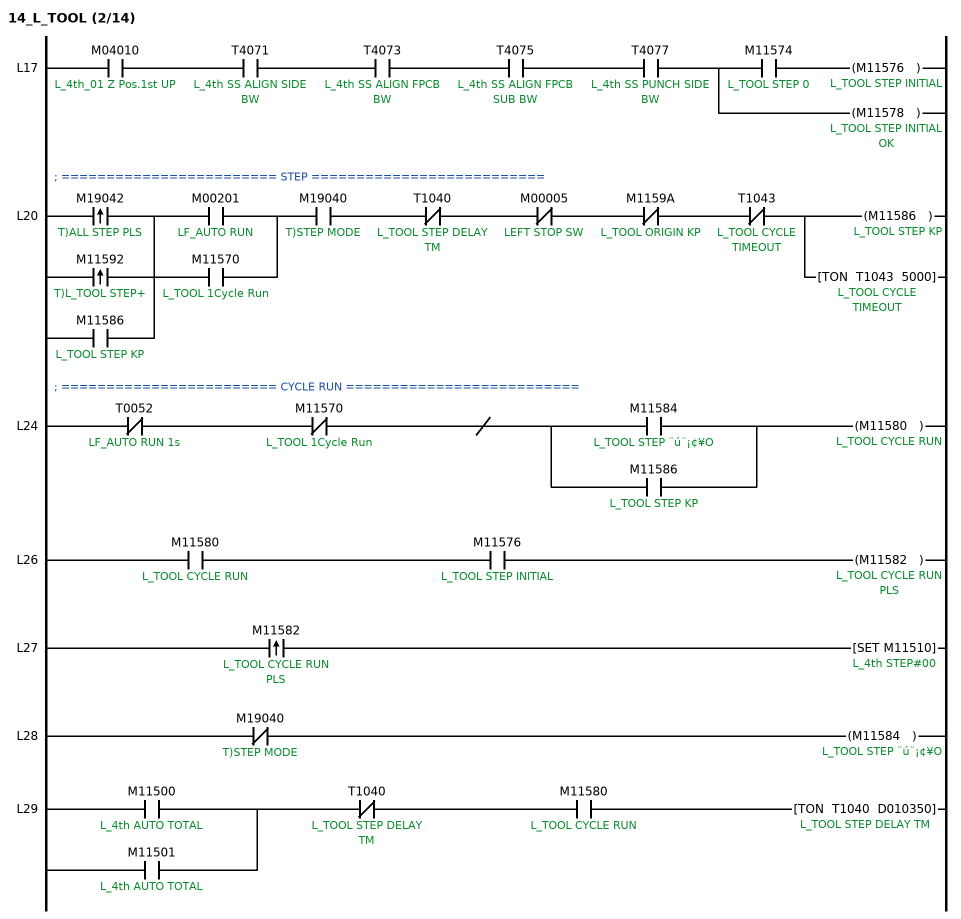
; L17
LOAD      M04010	// L_4th_01 Z Pos.1st UP
AND       T4071	// L_4th SS ALIGN SIDE BW
AND       T4073	// L_4th SS ALIGN FPCB BW
AND       T4075	// L_4th SS ALIGN FPCB SUB BW
AND       T4077	// L_4th SS PUNCH SIDE BW
MPUSH
AND       M11574	// L_TOOL STEP 0
OUT       M11576	// L_TOOL STEP INITIAL
MPOP
OUT       M11578	// L_TOOL STEP INITIAL OK
// ======================== STEP ==========================
; L20
LOADP     M19042	// T)ALL STEP PLS
ORP       M11592	// T)L_TOOL STEP+
OR        M11586	// L_TOOL STEP KP
LOAD      M00201	// LF_AUTO RUN
OR        M11570	// L_TOOL 1Cycle Run
AND LOAD
AND       M19040	// T)STEP MODE
AND NOT   T1040	// L_TOOL STEP DELAY TM
AND NOT   M00005	// LEFT STOP SW
AND NOT   M1159A	// L_TOOL ORIGIN KP
AND NOT   T1043	// L_TOOL CYCLE TIMEOUT
OUT       M11586	// L_TOOL STEP KP
TON       T1043 5000	// L_TOOL CYCLE TIMEOUT
// ======================== CYCLE RUN ==========================
; L24
LOAD NOT  T0052	// LF_AUTO RUN 1s
AND NOT   M11570	// L_TOOL 1Cycle Run
NOT
LOAD      M11584	// L_TOOL STEP ¨ú¨¡¢¥O
OR        M11586	// L_TOOL STEP KP
AND LOAD
OUT       M11580	// L_TOOL CYCLE RUN
; L26
LOAD      M11580	// L_TOOL CYCLE RUN
AND       M11576	// L_TOOL STEP INITIAL
OUT       M11582	// L_TOOL CYCLE RUN PLS
; L27
LOADP     M11582	// L_TOOL CYCLE RUN PLS
SET       M11510	// L_4th STEP#00
; L28
LOAD NOT  M19040	// T)STEP MODE
OUT       M11584	// L_TOOL STEP ¨ú¨¡¢¥O
; L29
LOAD      M11500	// L_4th AUTO TOTAL
OR        M11501	// L_4th AUTO TOTAL
AND NOT   T1040	// L_TOOL STEP DELAY TM
AND       M11580	// L_TOOL CYCLE RUN
TON       T1040 D010350	// L_TOOL STEP DELAY TM

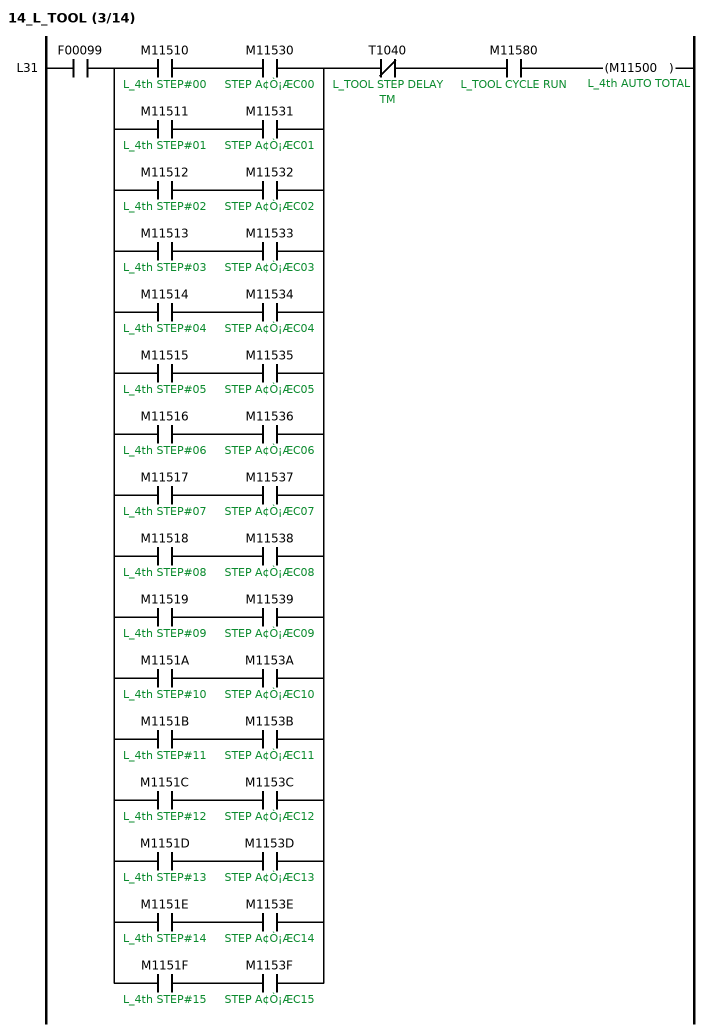
; L31
LOAD      F00099
LOAD      M11510	// L_4th STEP#00
AND       M11530	// STEP A¢Ò¡ÆC00
LOAD      M11511	// L_4th STEP#01
AND       M11531	// STEP A¢Ò¡ÆC01
OR LOAD
LOAD      M11512	// L_4th STEP#02
AND       M11532	// STEP A¢Ò¡ÆC02
OR LOAD
LOAD      M11513	// L_4th STEP#03
AND       M11533	// STEP A¢Ò¡ÆC03
OR LOAD
LOAD      M11514	// L_4th STEP#04
AND       M11534	// STEP A¢Ò¡ÆC04
OR LOAD
LOAD      M11515	// L_4th STEP#05
AND       M11535	// STEP A¢Ò¡ÆC05
OR LOAD
LOAD      M11516	// L_4th STEP#06
AND       M11536	// STEP A¢Ò¡ÆC06
OR LOAD
LOAD      M11517	// L_4th STEP#07
AND       M11537	// STEP A¢Ò¡ÆC07
OR LOAD
LOAD      M11518	// L_4th STEP#08
AND       M11538	// STEP A¢Ò¡ÆC08
OR LOAD
LOAD      M11519	// L_4th STEP#09
AND       M11539	// STEP A¢Ò¡ÆC09
OR LOAD
LOAD      M1151A	// L_4th STEP#10
AND       M1153A	// STEP A¢Ò¡ÆC10
OR LOAD
LOAD      M1151B	// L_4th STEP#11
AND       M1153B	// STEP A¢Ò¡ÆC11
OR LOAD
LOAD      M1151C	// L_4th STEP#12
AND       M1153C	// STEP A¢Ò¡ÆC12
OR LOAD
LOAD      M1151D	// L_4th STEP#13
AND       M1153D	// STEP A¢Ò¡ÆC13
OR LOAD
LOAD      M1151E	// L_4th STEP#14
AND       M1153E	// STEP A¢Ò¡ÆC14
OR LOAD
LOAD      M1151F	// L_4th STEP#15
AND       M1153F	// STEP A¢Ò¡ÆC15
OR LOAD
AND LOAD
AND NOT   T1040	// L_TOOL STEP DELAY TM
AND       M11580	// L_TOOL CYCLE RUN
OUT       M11500	// L_4th AUTO TOTAL

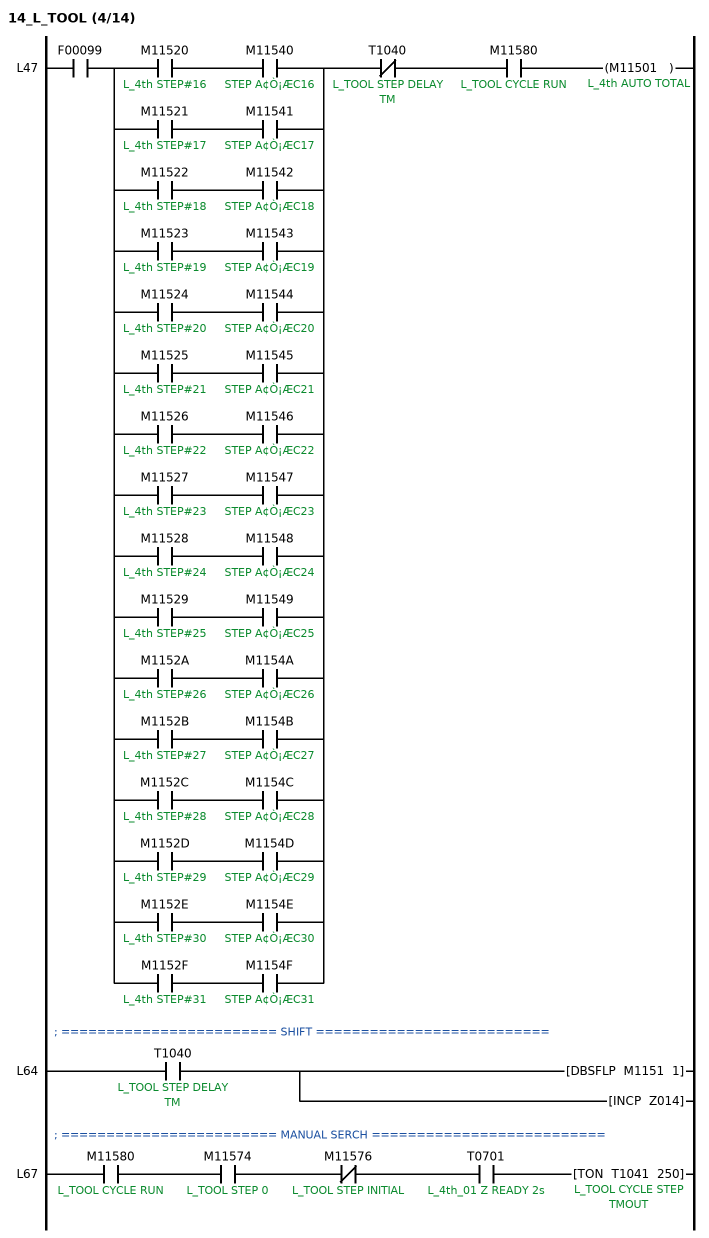
; L47
LOAD      F00099
LOAD      M11520	// L_4th STEP#16
AND       M11540	// STEP A¢Ò¡ÆC16
LOAD      M11521	// L_4th STEP#17
AND       M11541	// STEP A¢Ò¡ÆC17
OR LOAD
LOAD      M11522	// L_4th STEP#18
AND       M11542	// STEP A¢Ò¡ÆC18
OR LOAD
LOAD      M11523	// L_4th STEP#19
AND       M11543	// STEP A¢Ò¡ÆC19
OR LOAD
LOAD      M11524	// L_4th STEP#20
AND       M11544	// STEP A¢Ò¡ÆC20
OR LOAD
LOAD      M11525	// L_4th STEP#21
AND       M11545	// STEP A¢Ò¡ÆC21
OR LOAD
LOAD      M11526	// L_4th STEP#22
AND       M11546	// STEP A¢Ò¡ÆC22
OR LOAD
LOAD      M11527	// L_4th STEP#23
AND       M11547	// STEP A¢Ò¡ÆC23
OR LOAD
LOAD      M11528	// L_4th STEP#24
AND       M11548	// STEP A¢Ò¡ÆC24
OR LOAD
LOAD      M11529	// L_4th STEP#25
AND       M11549	// STEP A¢Ò¡ÆC25
OR LOAD
LOAD      M1152A	// L_4th STEP#26
AND       M1154A	// STEP A¢Ò¡ÆC26
OR LOAD
LOAD      M1152B	// L_4th STEP#27
AND       M1154B	// STEP A¢Ò¡ÆC27
OR LOAD
LOAD      M1152C	// L_4th STEP#28
AND       M1154C	// STEP A¢Ò¡ÆC28
OR LOAD
LOAD      M1152D	// L_4th STEP#29
AND       M1154D	// STEP A¢Ò¡ÆC29
OR LOAD
LOAD      M1152E	// L_4th STEP#30
AND       M1154E	// STEP A¢Ò¡ÆC30
OR LOAD
LOAD      M1152F	// L_4th STEP#31
AND       M1154F	// STEP A¢Ò¡ÆC31
OR LOAD
AND LOAD
AND NOT   T1040	// L_TOOL STEP DELAY TM
AND       M11580	// L_TOOL CYCLE RUN
OUT       M11501	// L_4th AUTO TOTAL
// ======================== SHIFT ==========================
; L64
LOAD      T1040	// L_TOOL STEP DELAY TM
DBSFLP    M1151 1
INCP      Z014
// ======================== MANUAL SERCH ==========================
; L67
LOAD      M11580	// L_TOOL CYCLE RUN
AND       M11574	// L_TOOL STEP 0
AND NOT   M11576	// L_TOOL STEP INITIAL
AND       T0701	// L_4th_01 Z READY 2s
TON       T1041 250	// L_TOOL CYCLE STEP TMOUT

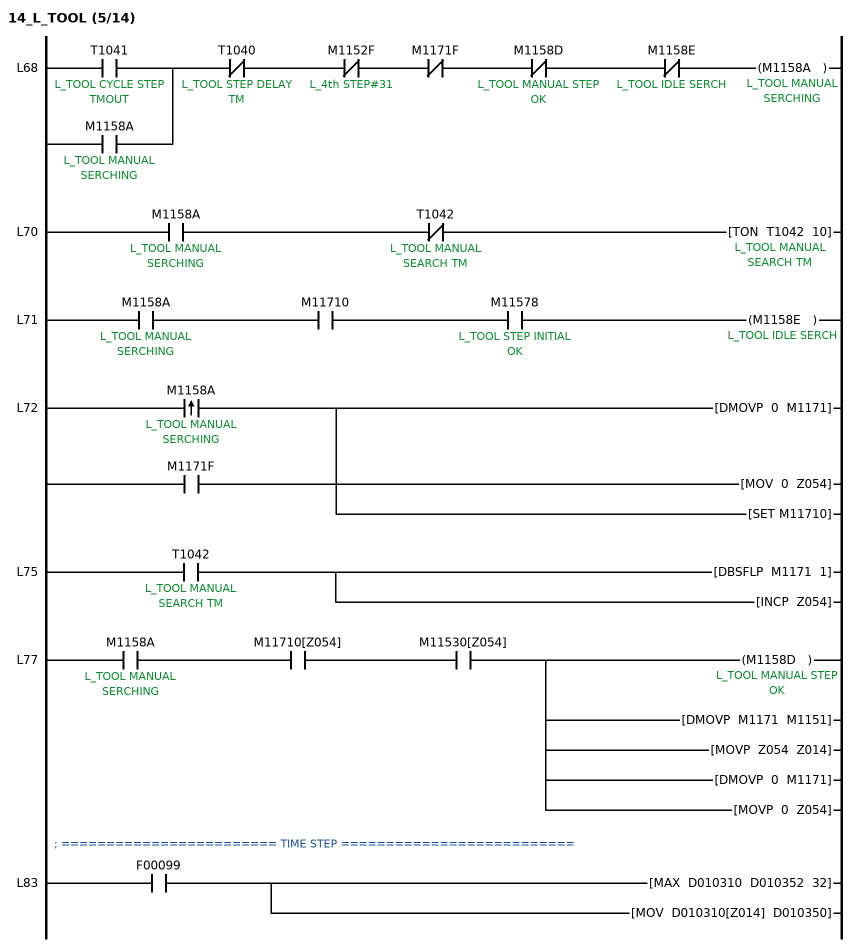
; L68
LOAD      T1041	// L_TOOL CYCLE STEP TMOUT
OR        M1158A	// L_TOOL MANUAL SERCHING
AND NOT   T1040	// L_TOOL STEP DELAY TM
AND NOT   M1152F	// L_4th STEP#31
AND NOT   M1171F
AND NOT   M1158D	// L_TOOL MANUAL STEP OK
AND NOT   M1158E	// L_TOOL IDLE SERCH
OUT       M1158A	// L_TOOL MANUAL SERCHING
; L70
LOAD      M1158A	// L_TOOL MANUAL SERCHING
AND NOT   T1042	// L_TOOL MANUAL SEARCH TM
TON       T1042 10	// L_TOOL MANUAL SEARCH TM
; L71
LOAD      M1158A	// L_TOOL MANUAL SERCHING
AND       M11710
AND       M11578	// L_TOOL STEP INITIAL OK
OUT       M1158E	// L_TOOL IDLE SERCH
; L72
LOADP     M1158A	// L_TOOL MANUAL SERCHING
OR        M1171F
DMOVP     0 M1171
MOV       0 Z054
SET       M11710
; L75
LOAD      T1042	// L_TOOL MANUAL SEARCH TM
DBSFLP    M1171 1
INCP      Z054
; L77
LOAD      M1158A	// L_TOOL MANUAL SERCHING
AND       M11710[Z054]
AND       M11530[Z054]
OUT       M1158D	// L_TOOL MANUAL STEP OK
DMOVP     M1171 M1151
MOVP      Z054 Z014
DMOVP     0 M1171
MOVP      0 Z054
// ======================== TIME STEP ==========================
; L83
LOAD      F00099
MAX       D010310 D010352 32
MOV       D010310[Z014] D010350

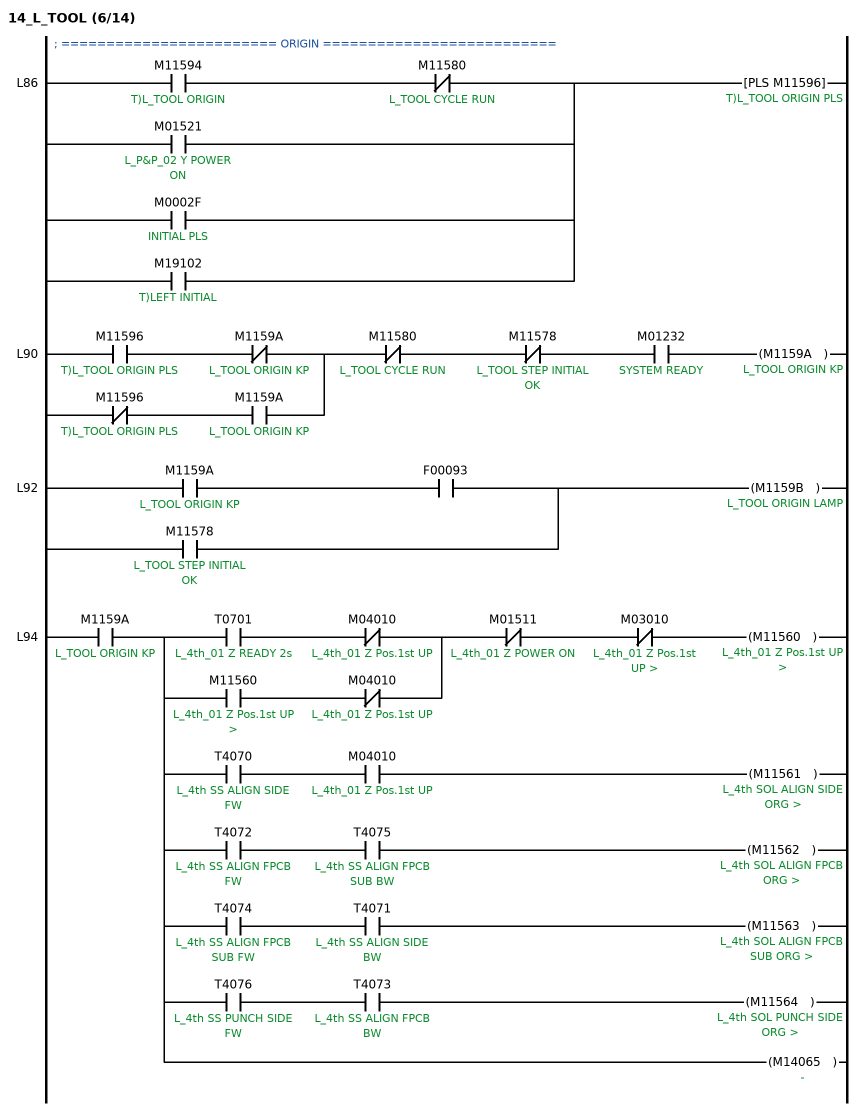
// ======================== ORIGIN ==========================
; L86
LOAD      M11594	// T)L_TOOL ORIGIN
AND NOT   M11580	// L_TOOL CYCLE RUN
OR        M01521	// L_P&P_02 Y POWER ON
OR        M0002F	// INITIAL PLS
OR        M19102	// T)LEFT INITIAL
OUTP      M11596	// T)L_TOOL ORIGIN PLS
; L90
LOAD      M11596	// T)L_TOOL ORIGIN PLS
AND NOT   M1159A	// L_TOOL ORIGIN KP
LOAD NOT  M11596	// T)L_TOOL ORIGIN PLS
AND       M1159A	// L_TOOL ORIGIN KP
OR LOAD
AND NOT   M11580	// L_TOOL CYCLE RUN
AND NOT   M11578	// L_TOOL STEP INITIAL OK
AND       M01232	// SYSTEM READY
OUT       M1159A	// L_TOOL ORIGIN KP
; L92
LOAD      M1159A	// L_TOOL ORIGIN KP
AND       F00093
OR        M11578	// L_TOOL STEP INITIAL OK
OUT       M1159B	// L_TOOL ORIGIN LAMP
; L94
LOAD      M1159A	// L_TOOL ORIGIN KP
MPUSH
LOAD      T0701	// L_4th_01 Z READY 2s
AND NOT   M04010	// L_4th_01 Z Pos.1st UP
LOAD      M11560	// L_4th_01 Z Pos.1st UP >
AND NOT   M04010	// L_4th_01 Z Pos.1st UP
OR LOAD
AND LOAD
AND NOT   M01511	// L_4th_01 Z POWER ON
AND NOT   M03010	// L_4th_01 Z Pos.1st     UP >
OUT       M11560	// L_4th_01 Z Pos.1st UP >
MLOAD
AND       T4070	// L_4th SS ALIGN SIDE FW
AND       M04010	// L_4th_01 Z Pos.1st UP
OUT       M11561	// L_4th SOL ALIGN SIDE ORG >
MLOAD
AND       T4072	// L_4th SS ALIGN FPCB FW
AND       T4075	// L_4th SS ALIGN FPCB SUB BW
OUT       M11562	// L_4th SOL ALIGN FPCB ORG >
MLOAD
AND       T4074	// L_4th SS ALIGN FPCB SUB FW
AND       T4071	// L_4th SS ALIGN SIDE BW
OUT       M11563	// L_4th SOL ALIGN FPCB SUB ORG >
MLOAD
AND       T4076	// L_4th SS PUNCH SIDE FW
AND       T4073	// L_4th SS ALIGN FPCB BW
OUT       M11564	// L_4th SOL PUNCH SIDE ORG >
MPOP
OUT       M14065	// -

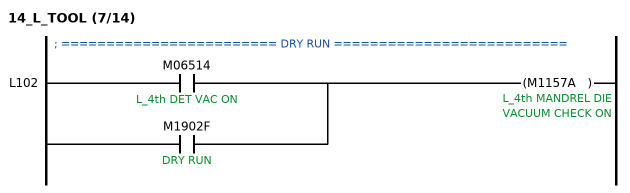
// ======================== DRY RUN ==========================
; L102
LOAD      M06514	// L_4th DET VAC ON
OR        M1902F	// DRY RUN
OUT       M1157A	// L_4th MANDREL DIE VACUUM CHECK ON

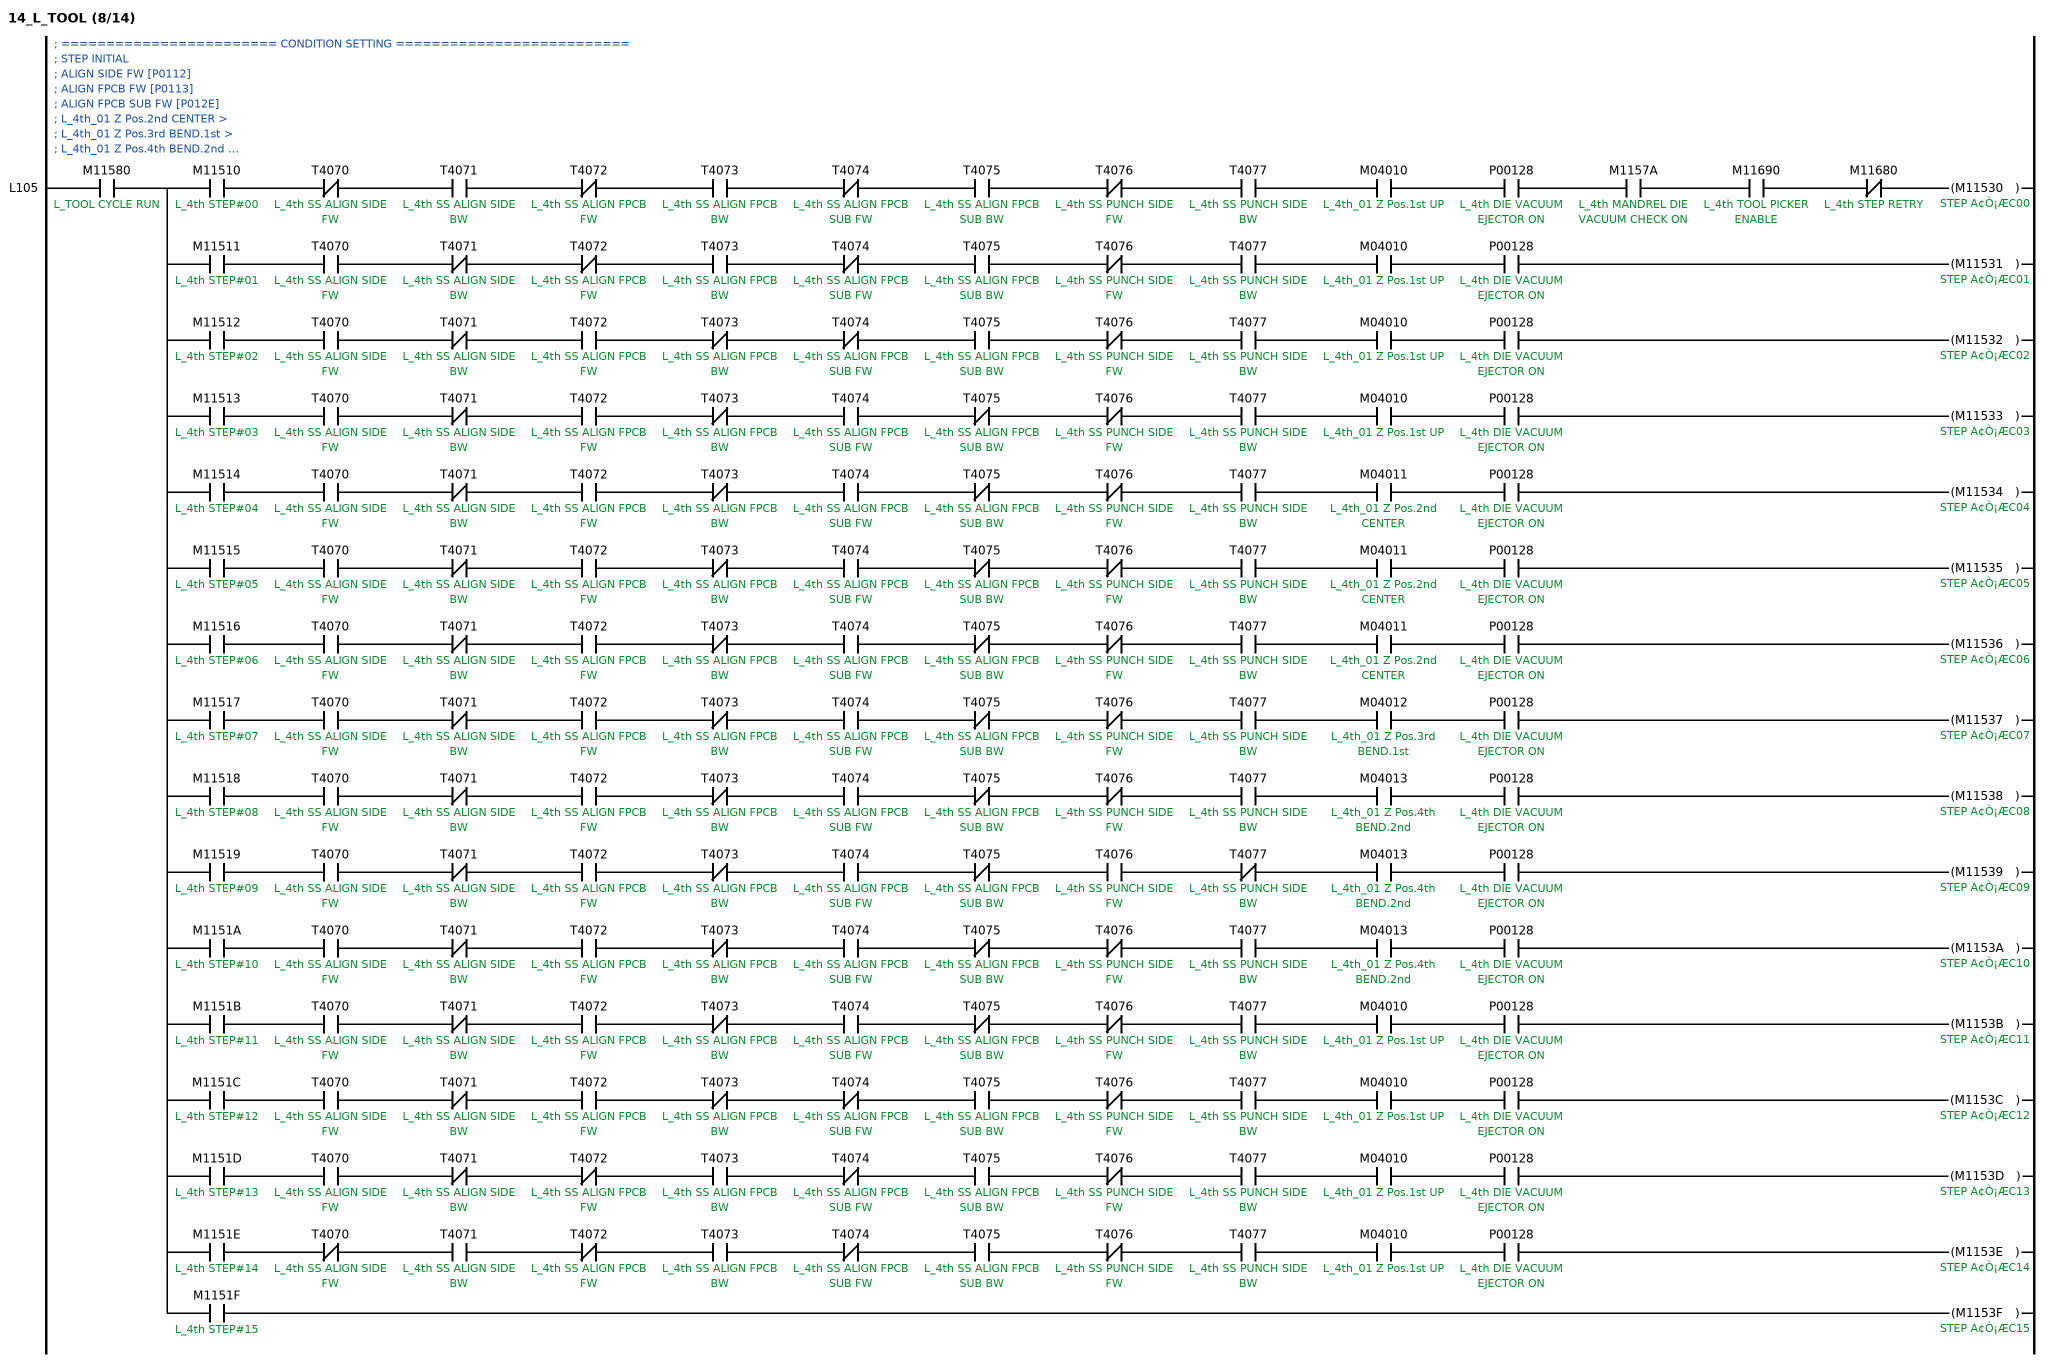
// ======================== CONDITION SETTING ==========================
; L105
LOAD      M11580	// L_TOOL CYCLE RUN
MPUSH
AND       M11510	// L_4th STEP#00
AND NOT   T4070	// L_4th SS ALIGN SIDE FW
AND       T4071	// L_4th SS ALIGN SIDE BW
AND NOT   T4072	// L_4th SS ALIGN FPCB FW
AND       T4073	// L_4th SS ALIGN FPCB BW
AND NOT   T4074	// L_4th SS ALIGN FPCB SUB FW
AND       T4075	// L_4th SS ALIGN FPCB SUB BW
AND NOT   T4076	// L_4th SS PUNCH SIDE FW
AND       T4077	// L_4th SS PUNCH SIDE BW
AND       M04010	// L_4th_01 Z Pos.1st UP
AND       P00128	// L_4th DIE VACUUM EJECTOR ON
AND       M1157A	// L_4th MANDREL DIE VACUUM CHECK ON
AND       M11690	// L_4th TOOL PICKER ENABLE
AND NOT   M11680	// L_4th STEP RETRY
OUT       M11530	// STEP A¢Ò¡ÆC00
MLOAD
AND       M11511	// L_4th STEP#01
AND       T4070	// L_4th SS ALIGN SIDE FW
AND NOT   T4071	// L_4th SS ALIGN SIDE BW
AND NOT   T4072	// L_4th SS ALIGN FPCB FW
AND       T4073	// L_4th SS ALIGN FPCB BW
AND NOT   T4074	// L_4th SS ALIGN FPCB SUB FW
AND       T4075	// L_4th SS ALIGN FPCB SUB BW
AND NOT   T4076	// L_4th SS PUNCH SIDE FW
AND       T4077	// L_4th SS PUNCH SIDE BW
AND       M04010	// L_4th_01 Z Pos.1st UP
AND       P00128	// L_4th DIE VACUUM EJECTOR ON
OUT       M11531	// STEP A¢Ò¡ÆC01
MLOAD
AND       M11512	// L_4th STEP#02
AND       T4070	// L_4th SS ALIGN SIDE FW
AND NOT   T4071	// L_4th SS ALIGN SIDE BW
AND       T4072	// L_4th SS ALIGN FPCB FW
AND NOT   T4073	// L_4th SS ALIGN FPCB BW
AND NOT   T4074	// L_4th SS ALIGN FPCB SUB FW
AND       T4075	// L_4th SS ALIGN FPCB SUB BW
AND NOT   T4076	// L_4th SS PUNCH SIDE FW
AND       T4077	// L_4th SS PUNCH SIDE BW
AND       M04010	// L_4th_01 Z Pos.1st UP
AND       P00128	// L_4th DIE VACUUM EJECTOR ON
OUT       M11532	// STEP A¢Ò¡ÆC02
MLOAD
AND       M11513	// L_4th STEP#03
AND       T4070	// L_4th SS ALIGN SIDE FW
AND NOT   T4071	// L_4th SS ALIGN SIDE BW
AND       T4072	// L_4th SS ALIGN FPCB FW
AND NOT   T4073	// L_4th SS ALIGN FPCB BW
AND       T4074	// L_4th SS ALIGN FPCB SUB FW
AND NOT   T4075	// L_4th SS ALIGN FPCB SUB BW
AND NOT   T4076	// L_4th SS PUNCH SIDE FW
AND       T4077	// L_4th SS PUNCH SIDE BW
AND       M04010	// L_4th_01 Z Pos.1st UP
AND       P00128	// L_4th DIE VACUUM EJECTOR ON
OUT       M11533	// STEP A¢Ò¡ÆC03
MLOAD
AND       M11514	// L_4th STEP#04
AND       T4070	// L_4th SS ALIGN SIDE FW
AND NOT   T4071	// L_4th SS ALIGN SIDE BW
AND       T4072	// L_4th SS ALIGN FPCB FW
AND NOT   T4073	// L_4th SS ALIGN FPCB BW
AND       T4074	// L_4th SS ALIGN FPCB SUB FW
AND NOT   T4075	// L_4th SS ALIGN FPCB SUB BW
AND NOT   T4076	// L_4th SS PUNCH SIDE FW
AND       T4077	// L_4th SS PUNCH SIDE BW
AND       M04011	// L_4th_01 Z Pos.2nd CENTER
AND       P00128	// L_4th DIE VACUUM EJECTOR ON
OUT       M11534	// STEP A¢Ò¡ÆC04
MLOAD
AND       M11515	// L_4th STEP#05
AND       T4070	// L_4th SS ALIGN SIDE FW
AND NOT   T4071	// L_4th SS ALIGN SIDE BW
AND       T4072	// L_4th SS ALIGN FPCB FW
AND NOT   T4073	// L_4th SS ALIGN FPCB BW
AND       T4074	// L_4th SS ALIGN FPCB SUB FW
AND NOT   T4075	// L_4th SS ALIGN FPCB SUB BW
AND NOT   T4076	// L_4th SS PUNCH SIDE FW
AND       T4077	// L_4th SS PUNCH SIDE BW
AND       M04011	// L_4th_01 Z Pos.2nd CENTER
AND       P00128	// L_4th DIE VACUUM EJECTOR ON
OUT       M11535	// STEP A¢Ò¡ÆC05
MLOAD
AND       M11516	// L_4th STEP#06
AND       T4070	// L_4th SS ALIGN SIDE FW
AND NOT   T4071	// L_4th SS ALIGN SIDE BW
AND       T4072	// L_4th SS ALIGN FPCB FW
AND NOT   T4073	// L_4th SS ALIGN FPCB BW
AND       T4074	// L_4th SS ALIGN FPCB SUB FW
AND NOT   T4075	// L_4th SS ALIGN FPCB SUB BW
AND NOT   T4076	// L_4th SS PUNCH SIDE FW
AND       T4077	// L_4th SS PUNCH SIDE BW
AND       M04011	// L_4th_01 Z Pos.2nd CENTER
AND       P00128	// L_4th DIE VACUUM EJECTOR ON
OUT       M11536	// STEP A¢Ò¡ÆC06
MLOAD
AND       M11517	// L_4th STEP#07
AND       T4070	// L_4th SS ALIGN SIDE FW
AND NOT   T4071	// L_4th SS ALIGN SIDE BW
AND       T4072	// L_4th SS ALIGN FPCB FW
AND NOT   T4073	// L_4th SS ALIGN FPCB BW
AND       T4074	// L_4th SS ALIGN FPCB SUB FW
AND NOT   T4075	// L_4th SS ALIGN FPCB SUB BW
AND NOT   T4076	// L_4th SS PUNCH SIDE FW
AND       T4077	// L_4th SS PUNCH SIDE BW
AND       M04012	// L_4th_01 Z Pos.3rd BEND.1st
AND       P00128	// L_4th DIE VACUUM EJECTOR ON
OUT       M11537	// STEP A¢Ò¡ÆC07
MLOAD
AND       M11518	// L_4th STEP#08
AND       T4070	// L_4th SS ALIGN SIDE FW
AND NOT   T4071	// L_4th SS ALIGN SIDE BW
AND       T4072	// L_4th SS ALIGN FPCB FW
AND NOT   T4073	// L_4th SS ALIGN FPCB BW
AND       T4074	// L_4th SS ALIGN FPCB SUB FW
AND NOT   T4075	// L_4th SS ALIGN FPCB SUB BW
AND NOT   T4076	// L_4th SS PUNCH SIDE FW
AND       T4077	// L_4th SS PUNCH SIDE BW
AND       M04013	// L_4th_01 Z Pos.4th BEND.2nd
AND       P00128	// L_4th DIE VACUUM EJECTOR ON
OUT       M11538	// STEP A¢Ò¡ÆC08
MLOAD
AND       M11519	// L_4th STEP#09
AND       T4070	// L_4th SS ALIGN SIDE FW
AND NOT   T4071	// L_4th SS ALIGN SIDE BW
AND       T4072	// L_4th SS ALIGN FPCB FW
AND NOT   T4073	// L_4th SS ALIGN FPCB BW
AND       T4074	// L_4th SS ALIGN FPCB SUB FW
AND NOT   T4075	// L_4th SS ALIGN FPCB SUB BW
AND       T4076	// L_4th SS PUNCH SIDE FW
AND NOT   T4077	// L_4th SS PUNCH SIDE BW
AND       M04013	// L_4th_01 Z Pos.4th BEND.2nd
AND       P00128	// L_4th DIE VACUUM EJECTOR ON
OUT       M11539	// STEP A¢Ò¡ÆC09
MLOAD
AND       M1151A	// L_4th STEP#10
AND       T4070	// L_4th SS ALIGN SIDE FW
AND NOT   T4071	// L_4th SS ALIGN SIDE BW
AND       T4072	// L_4th SS ALIGN FPCB FW
AND NOT   T4073	// L_4th SS ALIGN FPCB BW
AND       T4074	// L_4th SS ALIGN FPCB SUB FW
AND NOT   T4075	// L_4th SS ALIGN FPCB SUB BW
AND NOT   T4076	// L_4th SS PUNCH SIDE FW
AND       T4077	// L_4th SS PUNCH SIDE BW
AND       M04013	// L_4th_01 Z Pos.4th BEND.2nd
AND       P00128	// L_4th DIE VACUUM EJECTOR ON
OUT       M1153A	// STEP A¢Ò¡ÆC10
MLOAD
AND       M1151B	// L_4th STEP#11
AND       T4070	// L_4th SS ALIGN SIDE FW
AND NOT   T4071	// L_4th SS ALIGN SIDE BW
AND       T4072	// L_4th SS ALIGN FPCB FW
AND NOT   T4073	// L_4th SS ALIGN FPCB BW
AND       T4074	// L_4th SS ALIGN FPCB SUB FW
AND NOT   T4075	// L_4th SS ALIGN FPCB SUB BW
AND NOT   T4076	// L_4th SS PUNCH SIDE FW
AND       T4077	// L_4th SS PUNCH SIDE BW
AND       M04010	// L_4th_01 Z Pos.1st UP
AND       P00128	// L_4th DIE VACUUM EJECTOR ON
OUT       M1153B	// STEP A¢Ò¡ÆC11
MLOAD
AND       M1151C	// L_4th STEP#12
AND       T4070	// L_4th SS ALIGN SIDE FW
AND NOT   T4071	// L_4th SS ALIGN SIDE BW
AND       T4072	// L_4th SS ALIGN FPCB FW
AND NOT   T4073	// L_4th SS ALIGN FPCB BW
AND NOT   T4074	// L_4th SS ALIGN FPCB SUB FW
AND       T4075	// L_4th SS ALIGN FPCB SUB BW
AND NOT   T4076	// L_4th SS PUNCH SIDE FW
AND       T4077	// L_4th SS PUNCH SIDE BW
AND       M04010	// L_4th_01 Z Pos.1st UP
AND       P00128	// L_4th DIE VACUUM EJECTOR ON
OUT       M1153C	// STEP A¢Ò¡ÆC12
MLOAD
AND       M1151D	// L_4th STEP#13
AND       T4070	// L_4th SS ALIGN SIDE FW
AND NOT   T4071	// L_4th SS ALIGN SIDE BW
AND NOT   T4072	// L_4th SS ALIGN FPCB FW
AND       T4073	// L_4th SS ALIGN FPCB BW
AND NOT   T4074	// L_4th SS ALIGN FPCB SUB FW
AND       T4075	// L_4th SS ALIGN FPCB SUB BW
AND NOT   T4076	// L_4th SS PUNCH SIDE FW
AND       T4077	// L_4th SS PUNCH SIDE BW
AND       M04010	// L_4th_01 Z Pos.1st UP
AND       P00128	// L_4th DIE VACUUM EJECTOR ON
OUT       M1153D	// STEP A¢Ò¡ÆC13
MLOAD
AND       M1151E	// L_4th STEP#14
AND NOT   T4070	// L_4th SS ALIGN SIDE FW
AND       T4071	// L_4th SS ALIGN SIDE BW
AND NOT   T4072	// L_4th SS ALIGN FPCB FW
AND       T4073	// L_4th SS ALIGN FPCB BW
AND NOT   T4074	// L_4th SS ALIGN FPCB SUB FW
AND       T4075	// L_4th SS ALIGN FPCB SUB BW
AND NOT   T4076	// L_4th SS PUNCH SIDE FW
AND       T4077	// L_4th SS PUNCH SIDE BW
AND       M04010	// L_4th_01 Z Pos.1st UP
AND       P00128	// L_4th DIE VACUUM EJECTOR ON
OUT       M1153E	// STEP A¢Ò¡ÆC14
MPOP
AND       M1151F	// L_4th STEP#15
OUT       M1153F	// STEP A¢Ò¡ÆC15
// output comment: STEP INITIAL
// output comment: ALIGN SIDE FW [P0112]
// output comment: ALIGN FPCB FW [P0113]
// output comment: ALIGN FPCB SUB FW [P012E]
// output comment: L_4th_01 Z Pos.2nd CENTER >
// output comment: L_4th_01 Z Pos.3rd BEND.1st >
// output comment: L_4th_01 Z Pos.4th BEND.2nd >
// output comment: PUNCH SIDE FW [P012F]
// output comment: PUNCH SIDE BW [P012F]
// output comment: L_4th_01 Z Pos.1st       UP >
// output comment: ALIGN FPCB SUB BW [P012E]
// output comment: ALIGN FPCB BW [P0113]
// output comment: ALIGN SIDE BW   [P0112]

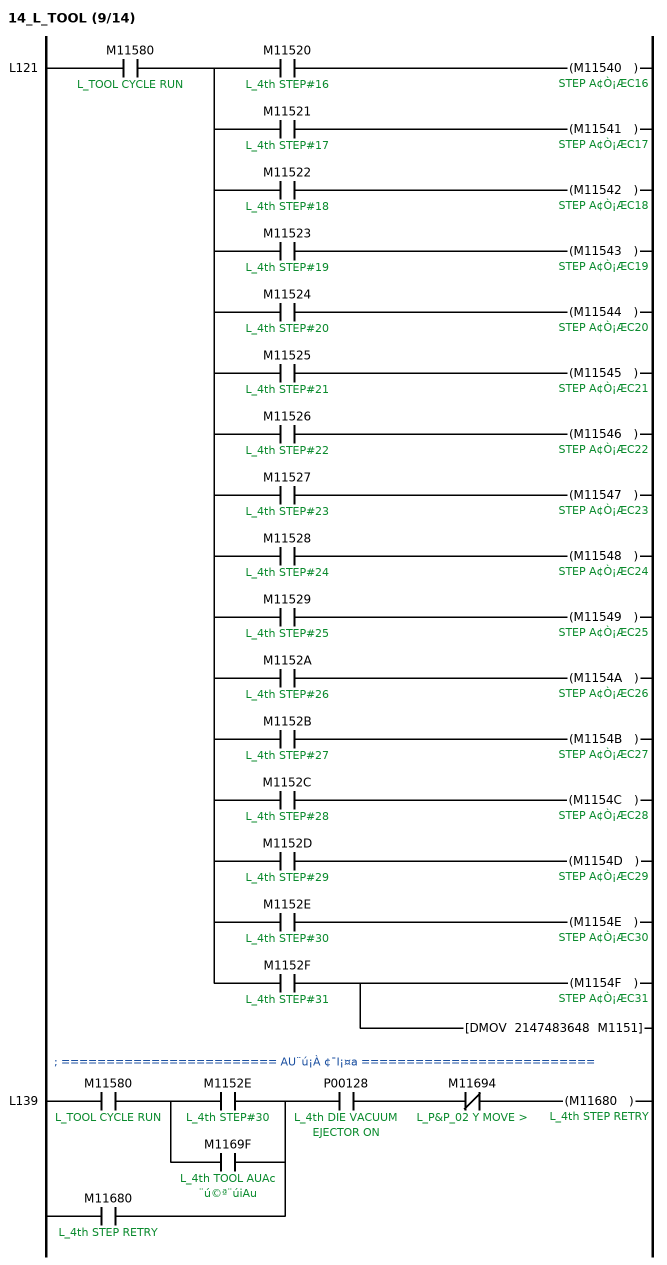
; L121
LOAD      M11580	// L_TOOL CYCLE RUN
MPUSH
AND       M11520	// L_4th STEP#16
OUT       M11540	// STEP A¢Ò¡ÆC16
MLOAD
AND       M11521	// L_4th STEP#17
OUT       M11541	// STEP A¢Ò¡ÆC17
MLOAD
AND       M11522	// L_4th STEP#18
OUT       M11542	// STEP A¢Ò¡ÆC18
MLOAD
AND       M11523	// L_4th STEP#19
OUT       M11543	// STEP A¢Ò¡ÆC19
MLOAD
AND       M11524	// L_4th STEP#20
OUT       M11544	// STEP A¢Ò¡ÆC20
MLOAD
AND       M11525	// L_4th STEP#21
OUT       M11545	// STEP A¢Ò¡ÆC21
MLOAD
AND       M11526	// L_4th STEP#22
OUT       M11546	// STEP A¢Ò¡ÆC22
MLOAD
AND       M11527	// L_4th STEP#23
OUT       M11547	// STEP A¢Ò¡ÆC23
MLOAD
AND       M11528	// L_4th STEP#24
OUT       M11548	// STEP A¢Ò¡ÆC24
MLOAD
AND       M11529	// L_4th STEP#25
OUT       M11549	// STEP A¢Ò¡ÆC25
MLOAD
AND       M1152A	// L_4th STEP#26
OUT       M1154A	// STEP A¢Ò¡ÆC26
MLOAD
AND       M1152B	// L_4th STEP#27
OUT       M1154B	// STEP A¢Ò¡ÆC27
MLOAD
AND       M1152C	// L_4th STEP#28
OUT       M1154C	// STEP A¢Ò¡ÆC28
MLOAD
AND       M1152D	// L_4th STEP#29
OUT       M1154D	// STEP A¢Ò¡ÆC29
MLOAD
AND       M1152E	// L_4th STEP#30
OUT       M1154E	// STEP A¢Ò¡ÆC30
MPOP
AND       M1152F	// L_4th STEP#31
OUT       M1154F	// STEP A¢Ò¡ÆC31
DMOV      2147483648 M1151
// ======================== AU¨ú¡À ¢¯I¡¤a ==========================
; L139
LOAD      M11580	// L_TOOL CYCLE RUN
LOAD      M1152E	// L_4th STEP#30
OR        M1169F	// L_4th TOOL AUAc ¨ú©ª¨úiAu
AND LOAD
OR        M11680	// L_4th STEP RETRY
AND       P00128	// L_4th DIE VACUUM EJECTOR ON
AND NOT   M11694	// L_P&P_02 Y MOVE >
OUT       M11680	// L_4th STEP RETRY

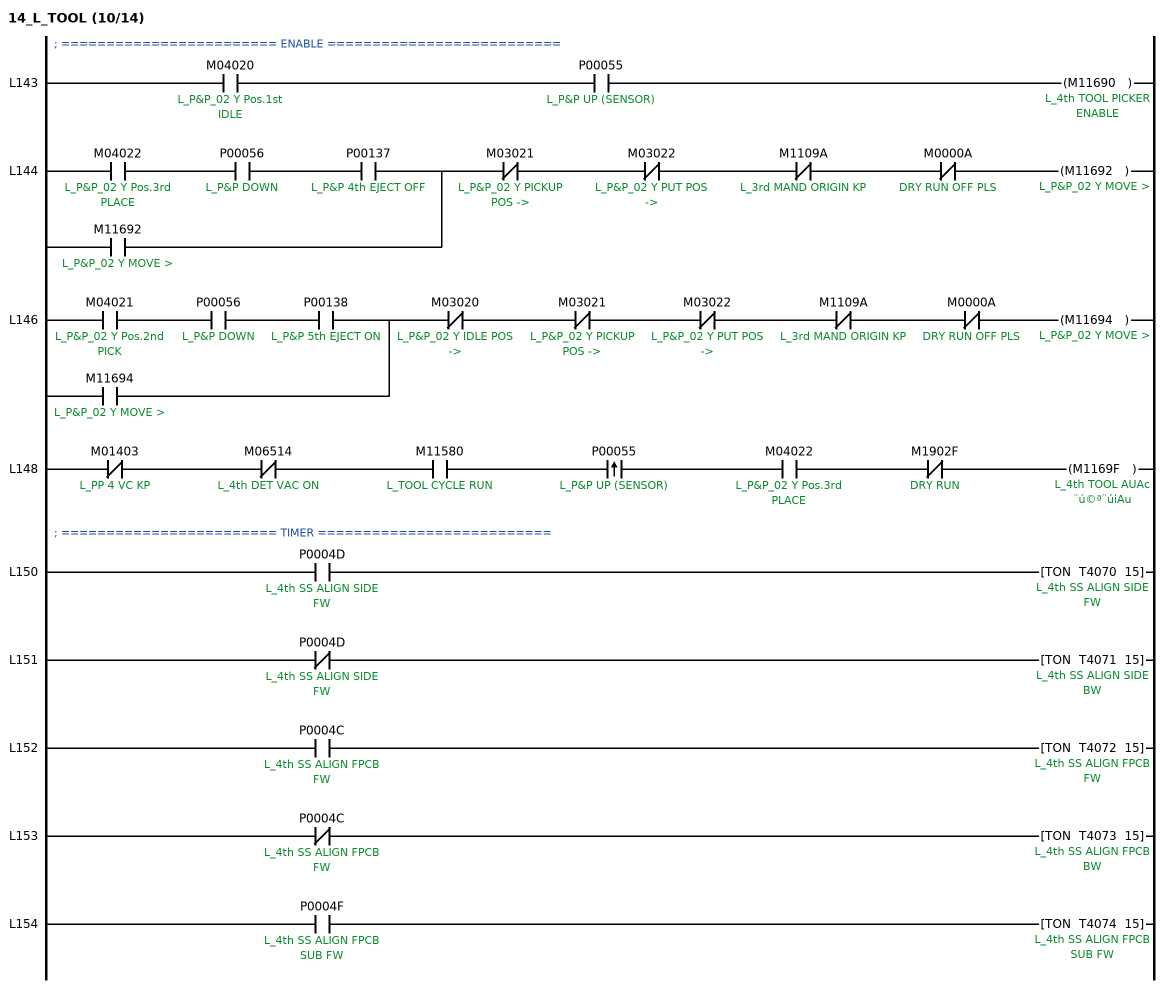
// ======================== ENABLE ==========================
; L143
LOAD      M04020	// L_P&P_02 Y Pos.1st IDLE
AND       P00055	// L_P&P UP (SENSOR)
OUT       M11690	// L_4th TOOL PICKER ENABLE
; L144
LOAD      M04022	// L_P&P_02 Y Pos.3rd PLACE
AND       P00056	// L_P&P DOWN
AND       P00137	// L_P&P 4th EJECT OFF
OR        M11692	// L_P&P_02 Y MOVE >
AND NOT   M03021	// L_P&P_02 Y PICKUP POS ->
AND NOT   M03022	// L_P&P_02 Y PUT POS ->
AND NOT   M1109A	// L_3rd MAND ORIGIN KP
AND NOT   M0000A	// DRY RUN OFF PLS
OUT       M11692	// L_P&P_02 Y MOVE >
; L146
LOAD      M04021	// L_P&P_02 Y Pos.2nd PICK
AND       P00056	// L_P&P DOWN
AND       P00138	// L_P&P 5th EJECT ON
OR        M11694	// L_P&P_02 Y MOVE >
AND NOT   M03020	// L_P&P_02 Y IDLE POS ->
AND NOT   M03021	// L_P&P_02 Y PICKUP POS ->
AND NOT   M03022	// L_P&P_02 Y PUT POS ->
AND NOT   M1109A	// L_3rd MAND ORIGIN KP
AND NOT   M0000A	// DRY RUN OFF PLS
OUT       M11694	// L_P&P_02 Y MOVE >
; L148
LOAD NOT  M01403	// L_PP 4 VC KP
AND NOT   M06514	// L_4th DET VAC ON
AND       M11580	// L_TOOL CYCLE RUN
ANDP      P00055	// L_P&P UP (SENSOR)
AND       M04022	// L_P&P_02 Y Pos.3rd PLACE
AND NOT   M1902F	// DRY RUN
OUT       M1169F	// L_4th TOOL AUAc ¨ú©ª¨úiAu
// ======================== TIMER ==========================
; L150
LOAD      P0004D	// L_4th SS ALIGN SIDE FW
TON       T4070 15	// L_4th SS ALIGN SIDE FW
; L151
LOAD NOT  P0004D	// L_4th SS ALIGN SIDE FW
TON       T4071 15	// L_4th SS ALIGN SIDE BW
; L152
LOAD      P0004C	// L_4th SS ALIGN FPCB FW
TON       T4072 15	// L_4th SS ALIGN FPCB FW
; L153
LOAD NOT  P0004C	// L_4th SS ALIGN FPCB FW
TON       T4073 15	// L_4th SS ALIGN FPCB BW
; L154
LOAD      P0004F	// L_4th SS ALIGN FPCB SUB FW
TON       T4074 15	// L_4th SS ALIGN FPCB SUB FW

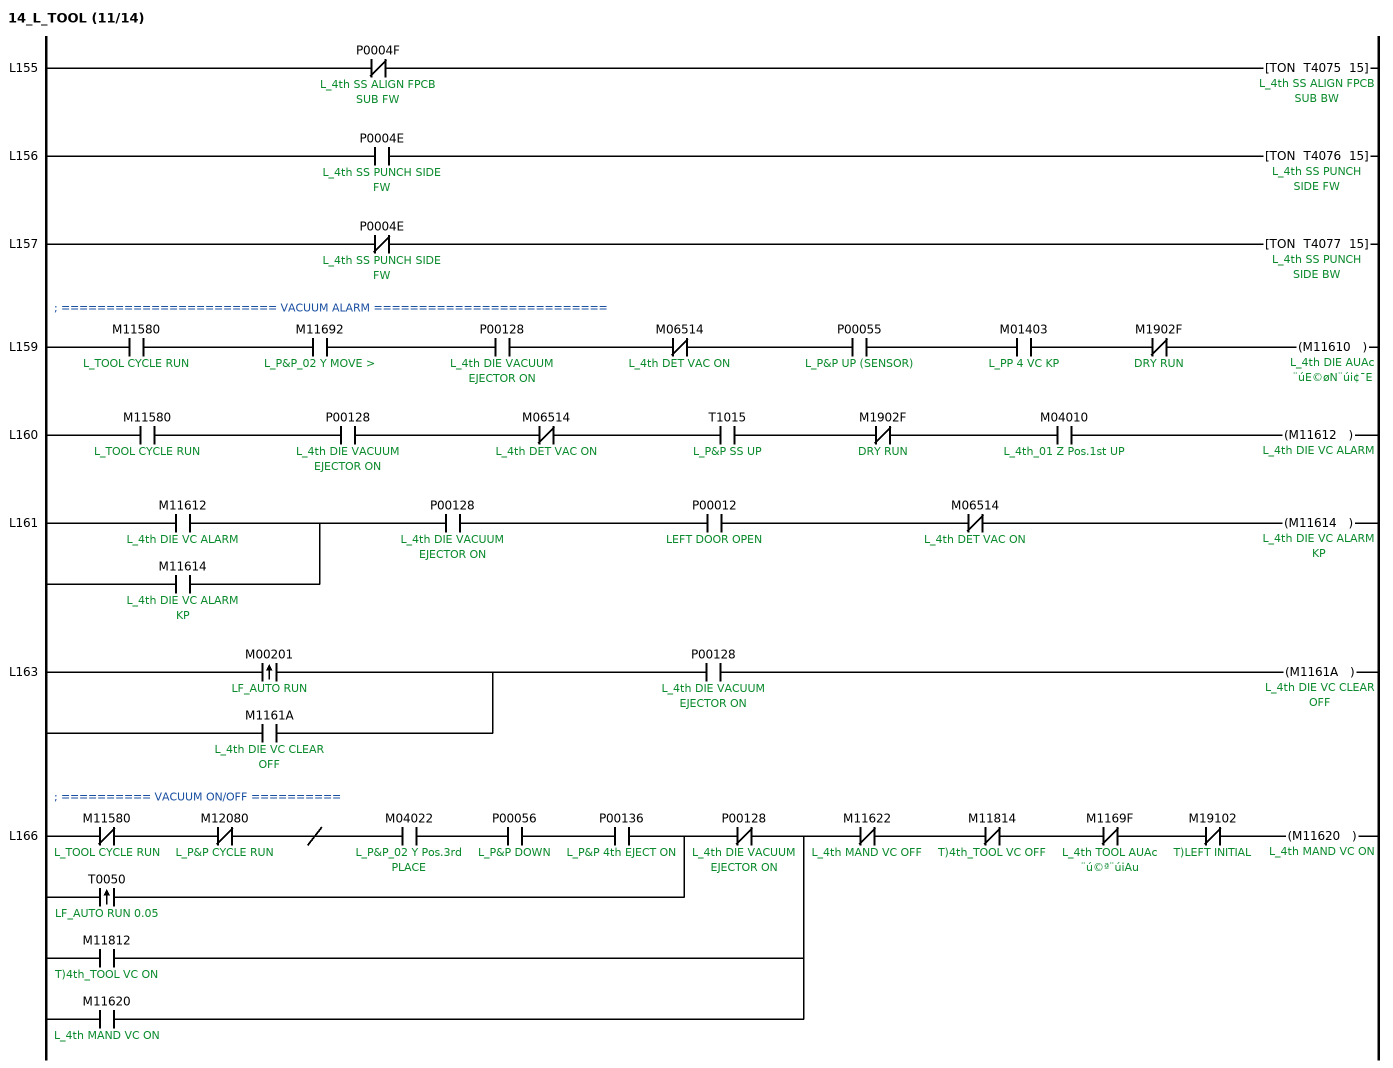
; L155
LOAD NOT  P0004F	// L_4th SS ALIGN FPCB SUB FW
TON       T4075 15	// L_4th SS ALIGN FPCB SUB BW
; L156
LOAD      P0004E	// L_4th SS PUNCH SIDE FW
TON       T4076 15	// L_4th SS PUNCH SIDE FW
; L157
LOAD NOT  P0004E	// L_4th SS PUNCH SIDE FW
TON       T4077 15	// L_4th SS PUNCH SIDE BW
// ======================== VACUUM ALARM ==========================
; L159
LOAD      M11580	// L_TOOL CYCLE RUN
AND       M11692	// L_P&P_02 Y MOVE >
AND       P00128	// L_4th DIE VACUUM EJECTOR ON
AND NOT   M06514	// L_4th DET VAC ON
AND       P00055	// L_P&P UP (SENSOR)
AND       M01403	// L_PP 4 VC KP
AND NOT   M1902F	// DRY RUN
OUT       M11610	// L_4th DIE AUAc ¨úE©øN¨úi¢¯E
; L160
LOAD      M11580	// L_TOOL CYCLE RUN
AND       P00128	// L_4th DIE VACUUM EJECTOR ON
AND NOT   M06514	// L_4th DET VAC ON
AND       T1015	// L_P&P SS UP
AND NOT   M1902F	// DRY RUN
AND       M04010	// L_4th_01 Z Pos.1st UP
OUT       M11612	// L_4th DIE VC ALARM
; L161
LOAD      M11612	// L_4th DIE VC ALARM
OR        M11614	// L_4th DIE VC ALARM KP
AND       P00128	// L_4th DIE VACUUM EJECTOR ON
AND       P00012	// LEFT DOOR OPEN
AND NOT   M06514	// L_4th DET VAC ON
OUT       M11614	// L_4th DIE VC ALARM KP
; L163
LOADP     M00201	// LF_AUTO RUN
OR        M1161A	// L_4th DIE VC CLEAR OFF
AND       P00128	// L_4th DIE VACUUM EJECTOR ON
OUT       M1161A	// L_4th DIE VC CLEAR OFF
// ========== VACUUM ON/OFF ==========
; L166
LOAD NOT  M11580	// L_TOOL CYCLE RUN
AND NOT   M12080	// L_P&P CYCLE RUN
NOT
AND       M04022	// L_P&P_02 Y Pos.3rd PLACE
AND       P00056	// L_P&P DOWN
AND       P00136	// L_P&P 4th EJECT ON
ORP       T0050	// LF_AUTO RUN 0.05
AND NOT   P00128	// L_4th DIE VACUUM EJECTOR ON
OR        M11812	// T)4th_TOOL VC ON
OR        M11620	// L_4th MAND VC ON
AND NOT   M11622	// L_4th MAND VC OFF
AND NOT   M11814	// T)4th_TOOL VC OFF
AND NOT   M1169F	// L_4th TOOL AUAc ¨ú©ª¨úiAu
AND NOT   M19102	// T)LEFT INITIAL
OUT       M11620	// L_4th MAND VC ON

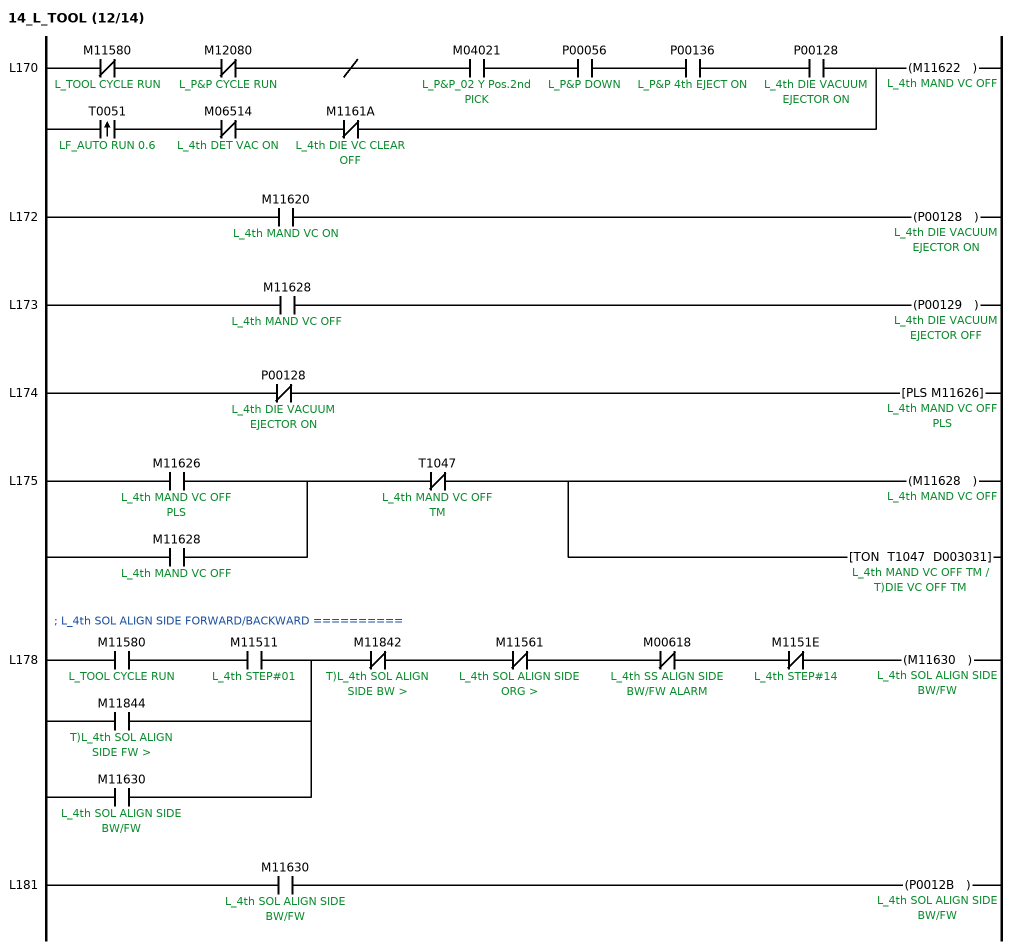
; L170
LOAD NOT  M11580	// L_TOOL CYCLE RUN
AND NOT   M12080	// L_P&P CYCLE RUN
NOT
AND       M04021	// L_P&P_02 Y Pos.2nd PICK
AND       P00056	// L_P&P DOWN
AND       P00136	// L_P&P 4th EJECT ON
AND       P00128	// L_4th DIE VACUUM EJECTOR ON
LOADP     T0051	// LF_AUTO RUN 0.6
AND NOT   M06514	// L_4th DET VAC ON
AND NOT   M1161A	// L_4th DIE VC CLEAR OFF
OR LOAD
OUT       M11622	// L_4th MAND VC OFF
; L172
LOAD      M11620	// L_4th MAND VC ON
OUT       P00128	// L_4th DIE VACUUM EJECTOR ON
; L173
LOAD      M11628	// L_4th MAND VC OFF
OUT       P00129	// L_4th DIE VACUUM EJECTOR OFF
; L174
LOAD NOT  P00128	// L_4th DIE VACUUM EJECTOR ON
OUTP      M11626	// L_4th MAND VC OFF PLS
; L175
LOAD      M11626	// L_4th MAND VC OFF PLS
OR        M11628	// L_4th MAND VC OFF
AND NOT   T1047	// L_4th MAND VC OFF TM
OUT       M11628	// L_4th MAND VC OFF
TON       T1047 D003031	// L_4th MAND VC OFF TM / T)DIE VC OFF TM
// L_4th SOL ALIGN SIDE FORWARD/BACKWARD ==========
; L178
LOAD      M11580	// L_TOOL CYCLE RUN
AND       M11511	// L_4th STEP#01
OR        M11844	// T)L_4th SOL ALIGN SIDE FW >
OR        M11630	// L_4th SOL ALIGN SIDE BW/FW
AND NOT   M11842	// T)L_4th SOL ALIGN SIDE BW >
AND NOT   M11561	// L_4th SOL ALIGN SIDE ORG >
AND NOT   M00618	// L_4th SS ALIGN SIDE BW/FW ALARM
AND NOT   M1151E	// L_4th STEP#14
OUT       M11630	// L_4th SOL ALIGN SIDE BW/FW
; L181
LOAD      M11630	// L_4th SOL ALIGN SIDE BW/FW
OUT       P0012B	// L_4th SOL ALIGN SIDE BW/FW

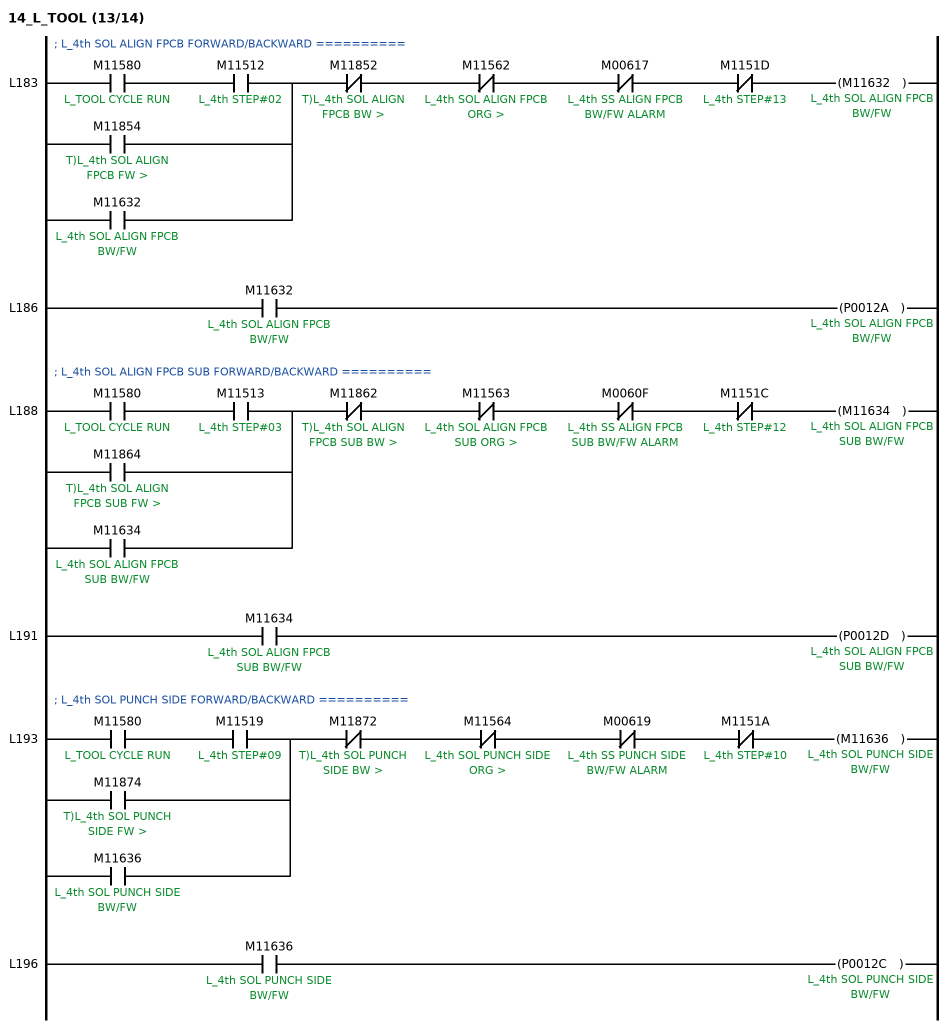
// L_4th SOL ALIGN FPCB FORWARD/BACKWARD ==========
; L183
LOAD      M11580	// L_TOOL CYCLE RUN
AND       M11512	// L_4th STEP#02
OR        M11854	// T)L_4th SOL ALIGN FPCB FW >
OR        M11632	// L_4th SOL ALIGN FPCB BW/FW
AND NOT   M11852	// T)L_4th SOL ALIGN FPCB BW >
AND NOT   M11562	// L_4th SOL ALIGN FPCB ORG >
AND NOT   M00617	// L_4th SS ALIGN FPCB BW/FW ALARM
AND NOT   M1151D	// L_4th STEP#13
OUT       M11632	// L_4th SOL ALIGN FPCB BW/FW
; L186
LOAD      M11632	// L_4th SOL ALIGN FPCB BW/FW
OUT       P0012A	// L_4th SOL ALIGN FPCB BW/FW
// L_4th SOL ALIGN FPCB SUB FORWARD/BACKWARD ==========
; L188
LOAD      M11580	// L_TOOL CYCLE RUN
AND       M11513	// L_4th STEP#03
OR        M11864	// T)L_4th SOL ALIGN FPCB SUB FW >
OR        M11634	// L_4th SOL ALIGN FPCB SUB BW/FW
AND NOT   M11862	// T)L_4th SOL ALIGN FPCB SUB BW >
AND NOT   M11563	// L_4th SOL ALIGN FPCB SUB ORG >
AND NOT   M0060F	// L_4th SS ALIGN FPCB SUB BW/FW ALARM
AND NOT   M1151C	// L_4th STEP#12
OUT       M11634	// L_4th SOL ALIGN FPCB SUB BW/FW
; L191
LOAD      M11634	// L_4th SOL ALIGN FPCB SUB BW/FW
OUT       P0012D	// L_4th SOL ALIGN FPCB SUB BW/FW
// L_4th SOL PUNCH SIDE FORWARD/BACKWARD ==========
; L193
LOAD      M11580	// L_TOOL CYCLE RUN
AND       M11519	// L_4th STEP#09
OR        M11874	// T)L_4th SOL PUNCH SIDE FW >
OR        M11636	// L_4th SOL PUNCH SIDE BW/FW
AND NOT   M11872	// T)L_4th SOL PUNCH SIDE BW >
AND NOT   M11564	// L_4th SOL PUNCH SIDE ORG >
AND NOT   M00619	// L_4th SS PUNCH SIDE BW/FW ALARM
AND NOT   M1151A	// L_4th STEP#10
OUT       M11636	// L_4th SOL PUNCH SIDE BW/FW
; L196
LOAD      M11636	// L_4th SOL PUNCH SIDE BW/FW
OUT       P0012C	// L_4th SOL PUNCH SIDE BW/FW

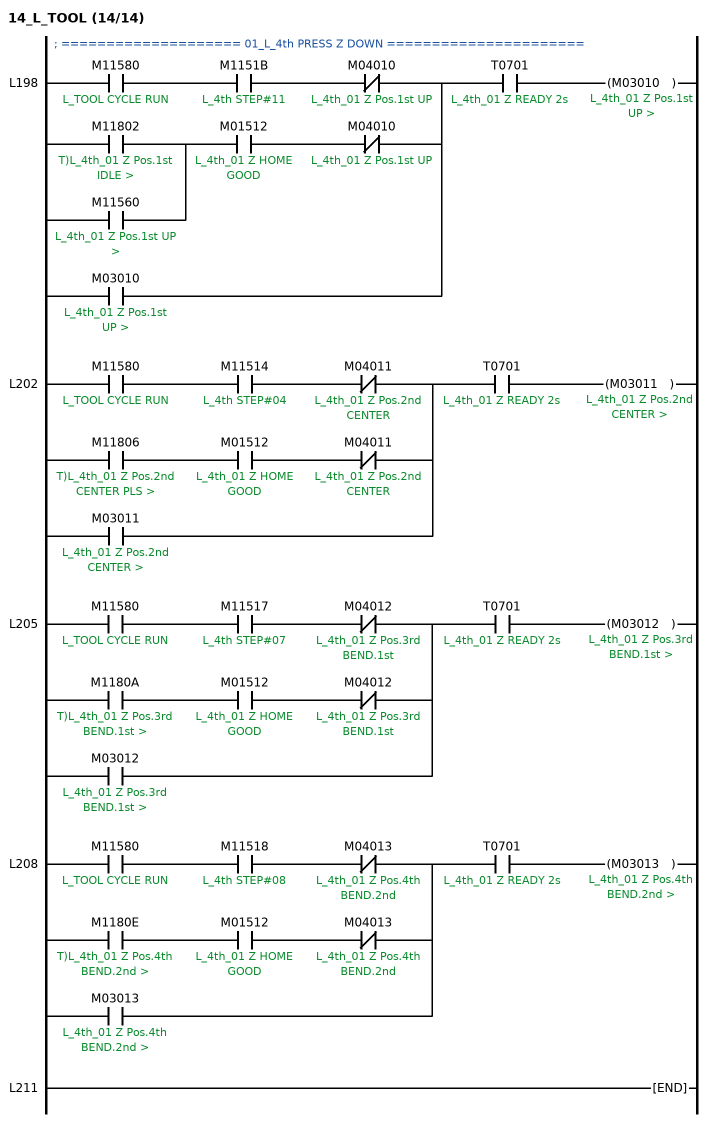
// ==================== 01_L_4th PRESS Z DOWN ======================
; L198
LOAD      M11580	// L_TOOL CYCLE RUN
AND       M1151B	// L_4th STEP#11
AND NOT   M04010	// L_4th_01 Z Pos.1st UP
LOAD      M11802	// T)L_4th_01 Z Pos.1st IDLE >
OR        M11560	// L_4th_01 Z Pos.1st UP >
AND       M01512	// L_4th_01 Z HOME GOOD
AND NOT   M04010	// L_4th_01 Z Pos.1st UP
OR LOAD
OR        M03010	// L_4th_01 Z Pos.1st     UP >
AND       T0701	// L_4th_01 Z READY 2s
OUT       M03010	// L_4th_01 Z Pos.1st     UP >
; L202
LOAD      M11580	// L_TOOL CYCLE RUN
AND       M11514	// L_4th STEP#04
AND NOT   M04011	// L_4th_01 Z Pos.2nd CENTER
LOAD      M11806	// T)L_4th_01 Z Pos.2nd CENTER PLS >
AND       M01512	// L_4th_01 Z HOME GOOD
AND NOT   M04011	// L_4th_01 Z Pos.2nd CENTER
OR LOAD
OR        M03011	// L_4th_01 Z Pos.2nd CENTER >
AND       T0701	// L_4th_01 Z READY 2s
OUT       M03011	// L_4th_01 Z Pos.2nd CENTER >
; L205
LOAD      M11580	// L_TOOL CYCLE RUN
AND       M11517	// L_4th STEP#07
AND NOT   M04012	// L_4th_01 Z Pos.3rd BEND.1st
LOAD      M1180A	// T)L_4th_01 Z Pos.3rd BEND.1st >
AND       M01512	// L_4th_01 Z HOME GOOD
AND NOT   M04012	// L_4th_01 Z Pos.3rd BEND.1st
OR LOAD
OR        M03012	// L_4th_01 Z Pos.3rd BEND.1st >
AND       T0701	// L_4th_01 Z READY 2s
OUT       M03012	// L_4th_01 Z Pos.3rd BEND.1st >
; L208
LOAD      M11580	// L_TOOL CYCLE RUN
AND       M11518	// L_4th STEP#08
AND NOT   M04013	// L_4th_01 Z Pos.4th BEND.2nd
LOAD      M1180E	// T)L_4th_01 Z Pos.4th BEND.2nd >
AND       M01512	// L_4th_01 Z HOME GOOD
AND NOT   M04013	// L_4th_01 Z Pos.4th BEND.2nd
OR LOAD
OR        M03013	// L_4th_01 Z Pos.4th BEND.2nd >
AND       T0701	// L_4th_01 Z READY 2s
OUT       M03013	// L_4th_01 Z Pos.4th BEND.2nd >
; L211
END

PROGRAM 15_L_PP (task: ½ºÄµ ÇÁ·Î±×·¥)

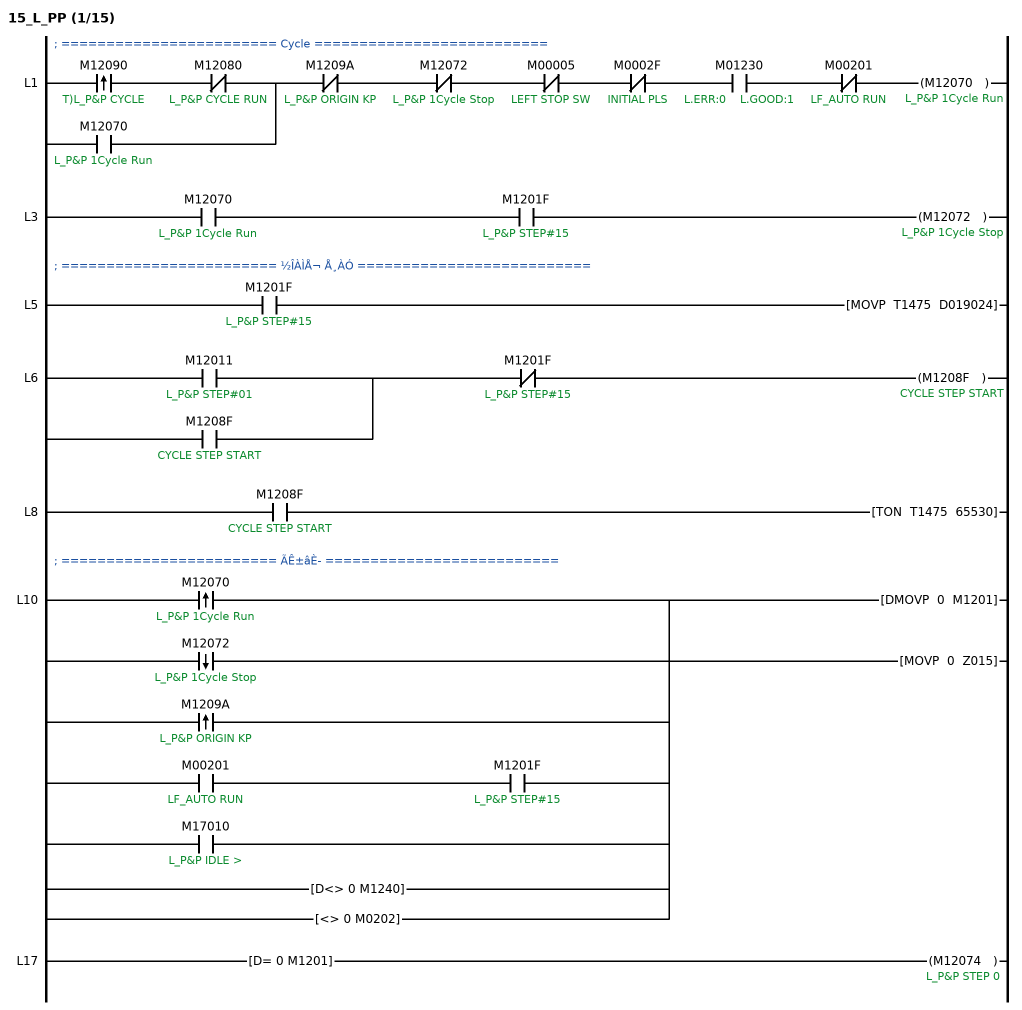
// ======================== Cycle ==========================
; L1
LOADP     M12090	// T)L_P&P CYCLE
AND NOT   M12080	// L_P&P CYCLE RUN
OR        M12070	// L_P&P 1Cycle Run
AND NOT   M1209A	// L_P&P ORIGIN KP
AND NOT   M12072	// L_P&P 1Cycle Stop
AND NOT   M00005	// LEFT STOP SW
AND NOT   M0002F	// INITIAL PLS
AND       M01230	// L.ERR:0    L.GOOD:1
AND NOT   M00201	// LF_AUTO RUN
OUT       M12070	// L_P&P 1Cycle Run
; L3
LOAD      M12070	// L_P&P 1Cycle Run
AND       M1201F	// L_P&P STEP#15
OUT       M12072	// L_P&P 1Cycle Stop
// ======================== ½ÎÀÌÅ¬ Å¸ÀÓ ==========================
; L5
LOAD      M1201F	// L_P&P STEP#15
MOVP      T1475 D019024
; L6
LOAD      M12011	// L_P&P STEP#01
OR        M1208F	// CYCLE STEP START
AND NOT   M1201F	// L_P&P STEP#15
OUT       M1208F	// CYCLE STEP START
; L8
LOAD      M1208F	// CYCLE STEP START
TON       T1475 65530
// ======================== ÃÊ±âÈ­ ==========================
; L10
LOADP     M12070	// L_P&P 1Cycle Run
ORN       M12072	// L_P&P 1Cycle Stop
ORP       M1209A	// L_P&P ORIGIN KP
LOAD      M00201	// LF_AUTO RUN
AND       M1201F	// L_P&P STEP#15
OR LOAD
OR        M17010	// L_P&P IDLE >
ORD<>     0 M1240
OR<>      0 M0202
DMOVP     0 M1201
MOVP      0 Z015
; L17
LOADD=    0 M1201
OUT       M12074	// L_P&P STEP 0

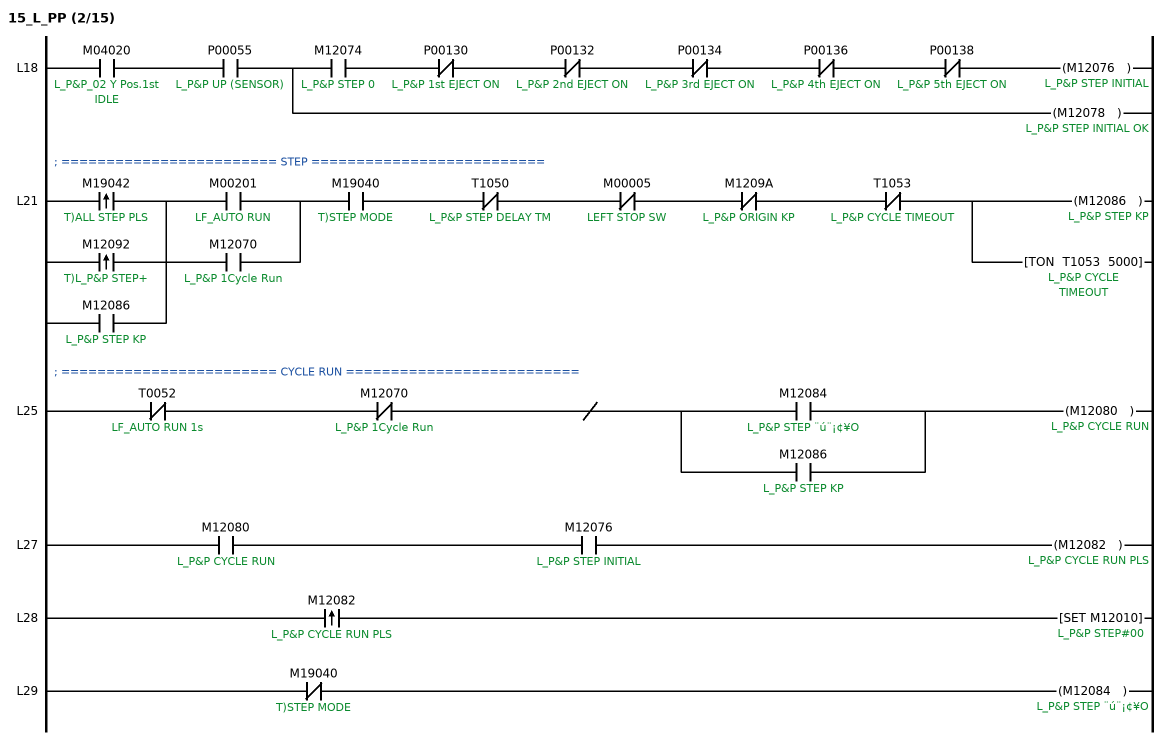
; L18
LOAD      M04020	// L_P&P_02 Y Pos.1st IDLE
AND       P00055	// L_P&P UP (SENSOR)
MPUSH
AND       M12074	// L_P&P STEP 0
AND NOT   P00130	// L_P&P 1st EJECT ON
AND NOT   P00132	// L_P&P 2nd EJECT ON
AND NOT   P00134	// L_P&P 3rd EJECT ON
AND NOT   P00136	// L_P&P 4th EJECT ON
AND NOT   P00138	// L_P&P 5th EJECT ON
OUT       M12076	// L_P&P STEP INITIAL
MPOP
OUT       M12078	// L_P&P STEP INITIAL OK
// ======================== STEP ==========================
; L21
LOADP     M19042	// T)ALL STEP PLS
ORP       M12092	// T)L_P&P STEP+
OR        M12086	// L_P&P STEP KP
LOAD      M00201	// LF_AUTO RUN
OR        M12070	// L_P&P 1Cycle Run
AND LOAD
AND       M19040	// T)STEP MODE
AND NOT   T1050	// L_P&P STEP DELAY TM
AND NOT   M00005	// LEFT STOP SW
AND NOT   M1209A	// L_P&P ORIGIN KP
AND NOT   T1053	// L_P&P CYCLE TIMEOUT
OUT       M12086	// L_P&P STEP KP
TON       T1053 5000	// L_P&P CYCLE TIMEOUT
// ======================== CYCLE RUN ==========================
; L25
LOAD NOT  T0052	// LF_AUTO RUN 1s
AND NOT   M12070	// L_P&P 1Cycle Run
NOT
LOAD      M12084	// L_P&P STEP ¨ú¨¡¢¥O
OR        M12086	// L_P&P STEP KP
AND LOAD
OUT       M12080	// L_P&P CYCLE RUN
; L27
LOAD      M12080	// L_P&P CYCLE RUN
AND       M12076	// L_P&P STEP INITIAL
OUT       M12082	// L_P&P CYCLE RUN PLS
; L28
LOADP     M12082	// L_P&P CYCLE RUN PLS
SET       M12010	// L_P&P STEP#00
; L29
LOAD NOT  M19040	// T)STEP MODE
OUT       M12084	// L_P&P STEP ¨ú¨¡¢¥O

